ABB RAPID module: Mov.mod

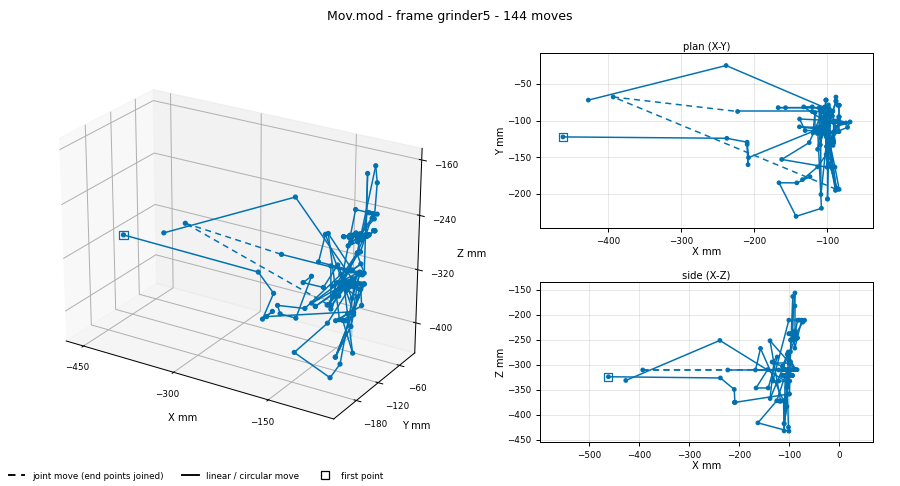
[picture p0: tool path of Mov.mod in frame grinder5, 144 of 396 moves have a stored position in this frame; points joined in program order, loops and branches not executed]
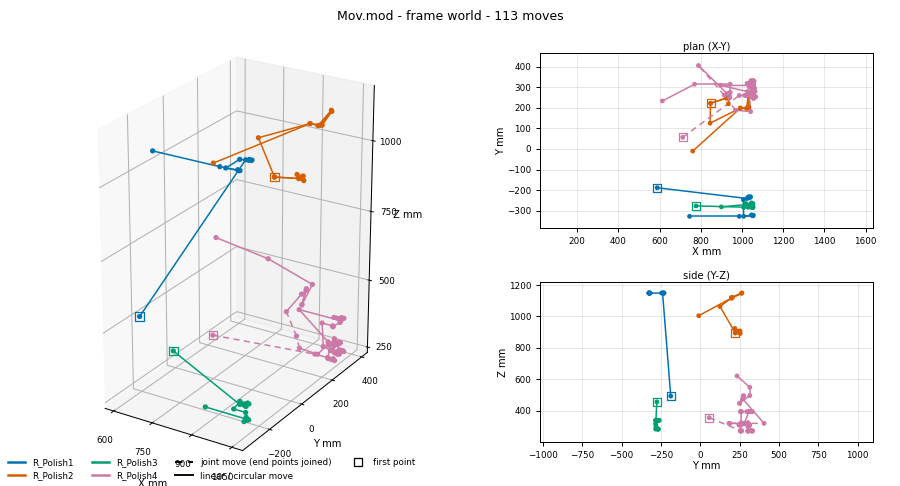
[picture p1: tool path of Mov.mod in frame world, 113 of 396 moves have a stored position in this frame; points joined in program order, loops and branches not executed]
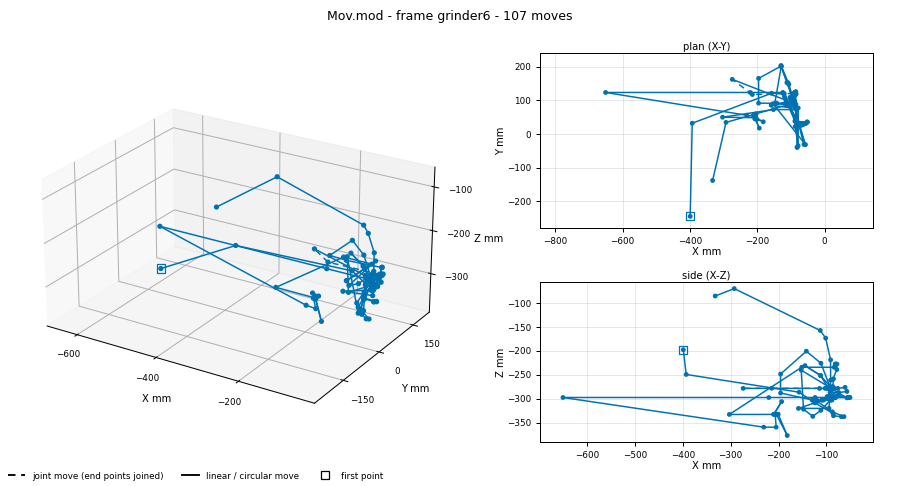
[picture p2: tool path of Mov.mod in frame grinder6, 107 of 396 moves have a stored position in this frame; points joined in program order, loops and branches not executed]
MODULE Mov

!******************************
! This program module for robot movements
! and storage of dynamic parameters
!******************************


! PALLET PARAMETERS
PERS num distance_p1_x:=60;
PERS num distance_p1_y:=160;
PERS num distance_p2_x:=60;
PERS num distance_p2_y:=160;

! DYNAMIC REGISTERS
PERS num loss_limit:=2;
PERS num collect:=1;
PERS num put:=1;
PERS num total:=0;
PERS num made:=0;
PERS num lost:=0;
PERS string start_data:="0000-00-00";

! TOOL DATA
PERS tooldata tool1:=[TRUE,[[0,0,320],[1,0,0,0]],[3,[0,0,130],[1,0,0,0],0,0,0]];
PERS tooldata tool2:=[TRUE,[[0,0,102],[1,0,0,0]],[3,[0,0,130],[1,0,0,0],0,0,0]];

TASK PERS tooldata a1:=[TRUE,[[0,0,344.1],[1,0,0,0]],[3,[0,0,130],[1,0,0,0],0,0,0]];
TASK PERS tooldata a2:=[TRUE,[[-72.3686,17.367,344.174],[1,0,0,0]],[3,[0,0,130],[1,0,0,0],0,0,0]];
TASK PERS tooldata a3:=[TRUE,[[-122,-5,344.174],[1,0,0,0]],[3,[0,0,130],[1,0,0,0],0,0,0]];
TASK PERS tooldata b1:=[TRUE,[[291.284,21.2677,171.248],[1,0,0,0]],[3,[70,0,130],[1,0,0,0],0,0,0]];

! WORK OBJECT DATA
PERS wobjdata pal1:=[FALSE,TRUE,"",[[760,-960,318],[4.81746E-05,-0.00506553,0.000941855,-0.999987]],[[540,0,0],[1,-9.27899E-07,1.32587E-06,-5.97185E-07]]];
PERS wobjdata pal2:=[FALSE,TRUE,"",[[149,-1059.8,461],[3.46326E-05,0.000526209,-0.000948043,0.999999]],[[0,0,0],[1,-3.72475E-06,5.79944E-06,-6.55528E-06]]];

TASK PERS wobjdata grinder1:=[FALSE,TRUE,"",[[1160.6,-280,1459],[1,0,0,0]],[[0,0,0],[1,0,0,0]]];
TASK PERS wobjdata grinder2:=[FALSE,TRUE,"",[[1160,280,1460],[1,0,0,0]],[[0,0,0],[1,0,0,0]]];
TASK PERS wobjdata grinder3:=[FALSE,TRUE,"",[[1156.5,-280,660],[1,0,0,0]],[[0,0,0],[1,0,0,0]]];
TASK PERS wobjdata grinder4:=[FALSE,TRUE,"",[[1158,280,656],[1,0,0,0]],[[6.65,0,-130],[1,0,0,0]]];
TASK PERS wobjdata grinder4_s:=[FALSE,TRUE,"",[[1157.8,510,518],[1,0,0,0]],[[0,0,0],[1,0,0,0]]];
TASK PERS wobjdata grinder5:=[FALSE,TRUE,"",[[280,1012,900],[0.70711,0,0,0.70711]],[[0,0,0],[1,0,0,0]]];
TASK PERS wobjdata grinder6:=[FALSE,TRUE,"",[[-282,1000,900],[0.70711,0,0,0.70711]],[[0,0,0],[1,0,0,0]]];

! POSITIONS
PERS robtarget home:=[[649.18,-0.03,789.42],[2.73078E-05,2.31734E-05,1,2.09338E-05],[-1,0,-1,0],[9E+09,9E+09,9E+09,9E+09,9E+09,9E+09]];
PERS robtarget corner:=[[286.64,-742.95,588.29],[0.00624253,-0.703358,-0.710805,0.00220458],[-1,-1,0,0],[9E+09,9E+09,9E+09,9E+09,9E+09,9E+09]];
PERS robtarget before:=[[683.43,-725.72,546.02],[0.0245473,-0.706641,-0.706937,-0.0172306],[-1,0,0,0],[9E+09,9E+09,9E+09,9E+09,9E+09,9E+09]];
PERS robtarget check:=[[764.25,-750.95,502.27],[0.0244543,-0.706556,-0.707026,-0.017169],[-1,0,0,0],[9E+09,9E+09,9E+09,9E+09,9E+09,9E+09]];
PERS robtarget after:=[[683.45,-725.70,546.02],[0.0245494,-0.706651,-0.706925,-0.0172644],[-1,0,0,0],[9E+09,9E+09,9E+09,9E+09,9E+09,9E+09]];
PERS robtarget non_drop:=[[286.65,-1103.34,974.46],[0.311182,0.630793,0.633652,-0.322103],[-1,-1,0,0],[9E+9,9E+9,9E+9,9E+9,9E+9,9E+9]];

PERS robtarget wheel5:=[[-112.72,-79.92,-299.81],[0.228521,0.250847,0.938723,-0.0604406],[0,-1,0,0],[9E+09,9E+09,9E+09,9E+09,9E+09,9E+09]];
PERS robtarget wheel6:=[[-100.57,98.49,-299.81],[0.221539,0.223786,0.947859,0.0490301],[1,-1,0,0],[9E+09,9E+09,9E+09,9E+09,9E+09,9E+09]];

! OFFSET PARAMETER
PERS num count5:=0;
PERS num count6:=0;
PERS num count5_limit:=1700;
PERS num count6_limit:=1700;

PERS num offs5_step:=0.01;
PERS num offs6_step:=0.01;


!******************************
PROC P_Parameters()
    distance_p1_x:=60;
    distance_p1_y:=160;
    distance_p2_x:=60;
    distance_p2_y:=160;
ENDPROC

!******************************
PROC R_Take1()
    Set DO10_60;
    !
    MoveL [[81.54,-63.78,264.56],[0.00371365,0.713716,-0.700414,0.00397575],[-1,-1,0,0],[9E+09,9E+09,9E+09,9E+09,9E+09,9E+09]],s500,z50,tool1\WObj:=pal1;
    MoveL [[79.44,-63.69,183.91],[0.011189,0.710235,-0.703782,0.0114969],[-1,0,0,0],[9E+09,9E+09,9E+09,9E+09,9E+09,9E+09]],s100,z10,tool1\WObj:=pal1;
    MoveL [[80.22,-63.55,118.78],[0.00697535,0.710341,-0.703813,0.00376915],[-1,0,0,0],[9E+09,9E+09,9E+09,9E+09,9E+09,9E+09]],s50,fine,tool1\WObj:=pal1;
    MoveL [[78.90,-63.58,118.50],[0.0118877,0.702177,-0.71189,-0.00426993],[-1,0,0,0],[9E+09,9E+09,9E+09,9E+09,9E+09,9E+09]],s25,fine,tool1\WObj:=pal1;
    MoveL [[78.90,-63.55,117.64],[0.00382538,0.726156,-0.687509,0.00387196],[-1,-1,0,0],[9E+09,9E+09,9E+09,9E+09,9E+09,9E+09]],s25,fine,tool1\WObj:=pal1;
    MoveL [[80.70,-63.58,116.47],[0.00384294,0.724898,-0.688834,0.00390763],[-1,-1,0,0],[9E+09,9E+09,9E+09,9E+09,9E+09,9E+09]],s25,fine,tool1\WObj:=pal1;
    !
    T_Grab;
    !
    MoveL [[81.00,-63.59,147.58],[0.0127632,0.716524,-0.697325,0.0129917],[-1,0,0,0],[9E+09,9E+09,9E+09,9E+09,9E+09,9E+09]],s50,fine,tool1\WObj:=pal1;
    MoveL [[81.31,-63.65,178.40],[0.0171099,0.716402,-0.69726,0.0174624],[-1,0,0,0],[9E+09,9E+09,9E+09,9E+09,9E+09,9E+09]],s150,z5,tool1\WObj:=pal1;
    MoveL [[81.48,-63.80,264.59],[0.00373939,0.713705,-0.700425,0.00394878],[-1,-1,0,0],[9E+09,9E+09,9E+09,9E+09,9E+09,9E+09]],s500,z50,tool1\WObj:=pal1;
ENDPROC

!******************************
PROC R_Take2()
    MoveL [[81.54,-63.78,264.56],[0.00371365,0.713716,-0.700414,0.00397575],[-1,-1,0,0],[9E+09,9E+09,9E+09,9E+09,9E+09,9E+09]],s500,z50,tool1\WObj:=pal1;
    MoveL [[79.44,-63.69,183.91],[0.011189,0.710235,-0.703782,0.0114969],[-1,0,0,0],[9E+09,9E+09,9E+09,9E+09,9E+09,9E+09]],s100,z10,tool1\WObj:=pal1;
    MoveL [[80.22,-63.55,118.78],[0.00697535,0.710341,-0.703813,0.00376915],[-1,0,0,0],[9E+09,9E+09,9E+09,9E+09,9E+09,9E+09]],s50,fine,tool1\WObj:=pal1;
    MoveL [[78.90,-63.58,118.50],[0.0118877,0.702177,-0.71189,-0.00426993],[-1,0,0,0],[9E+09,9E+09,9E+09,9E+09,9E+09,9E+09]],s25,fine,tool1\WObj:=pal1;
    MoveL [[78.90,-63.55,117.64],[0.00382538,0.726156,-0.687509,0.00387196],[-1,-1,0,0],[9E+09,9E+09,9E+09,9E+09,9E+09,9E+09]],s25,fine,tool1\WObj:=pal1;
    MoveL [[80.70,-63.58,116.47],[0.00384294,0.724898,-0.688834,0.00390763],[-1,-1,0,0],[9E+09,9E+09,9E+09,9E+09,9E+09,9E+09]],s25,fine,tool1\WObj:=pal1;
    !
    T_Grab;
    !
    MoveL [[81.00,-63.59,147.58],[0.0127632,0.716524,-0.697325,0.0129917],[-1,0,0,0],[9E+09,9E+09,9E+09,9E+09,9E+09,9E+09]],s50,fine,tool1\WObj:=pal1;
    MoveL [[81.31,-63.65,178.40],[0.0171099,0.716402,-0.69726,0.0174624],[-1,0,0,0],[9E+09,9E+09,9E+09,9E+09,9E+09,9E+09]],s150,z5,tool1\WObj:=pal1;
    MoveL [[81.48,-63.80,264.59],[0.00373939,0.713705,-0.700425,0.00394878],[-1,-1,0,0],[9E+09,9E+09,9E+09,9E+09,9E+09,9E+09]],s500,z50,tool1\WObj:=pal1;
ENDPROC

!******************************
PROC R_Drop1()
    MoveL [[81.49,-63.80,264.52],[0.00378181,0.713658,-0.700473,0.0039678],[-1,-1,0,0],[9E+09,9E+09,9E+09,9E+09,9E+09,9E+09]],s500,z50,tool1\WObj:=pal1;
    MoveL [[81.16,-63.64,177.38],[0.015051,0.720309,-0.693317,0.0154864],[-1,0,0,0],[9E+09,9E+09,9E+09,9E+09,9E+09,9E+09]],s500,z10,tool1\WObj:=pal1;
    MoveL [[80.98,-63.98,149.80],[0.0150862,0.715998,-0.697765,0.0155745],[-1,0,0,0],[9E+09,9E+09,9E+09,9E+09,9E+09,9E+09]],s100,z1,tool1\WObj:=pal1;
    MoveL [[79.99,-63.75,138.99],[0.0152028,0.720859,-0.692742,0.0154934],[-1,0,0,0],[9E+09,9E+09,9E+09,9E+09,9E+09,9E+09]],s50,fine,tool1\WObj:=pal1;
    !
    T_Release;
    !
    MoveL [[80.08,-63.90,158.90],[0.0175743,0.722459,-0.690952,0.0181282],[-1,0,0,0],[9E+09,9E+09,9E+09,9E+09,9E+09,9E+09]],s20,fine,tool1\WObj:=pal1;
    MoveL [[81.01,-63.73,207.27],[0.00381861,0.72049,-0.693443,0.00397601],[-1,-1,0,0],[9E+09,9E+09,9E+09,9E+09,9E+09,9E+09]],s50,z50,tool1\WObj:=pal1;
    MoveL [[81.54,-63.77,264.48],[0.00376586,0.713646,-0.700485,0.00398274],[-1,-1,0,0],[9E+09,9E+09,9E+09,9E+09,9E+09,9E+09]],s500,z50,tool1\WObj:=pal1;
    !
    Reset DO10_60;
ENDPROC

!******************************
PROC R_Drop2()
    MoveL [[81.49,-63.80,264.52],[0.00378181,0.713658,-0.700473,0.0039678],[-1,-1,0,0],[9E+09,9E+09,9E+09,9E+09,9E+09,9E+09]],s500,z50,tool1\WObj:=pal1;
    MoveL [[81.16,-63.64,177.38],[0.015051,0.720309,-0.693317,0.0154864],[-1,0,0,0],[9E+09,9E+09,9E+09,9E+09,9E+09,9E+09]],s500,z10,tool1\WObj:=pal1;
    MoveL [[80.98,-63.98,149.80],[0.0150862,0.715998,-0.697765,0.0155745],[-1,0,0,0],[9E+09,9E+09,9E+09,9E+09,9E+09,9E+09]],s100,z1,tool1\WObj:=pal1;
    MoveL [[79.99,-63.75,138.99],[0.0152028,0.720859,-0.692742,0.0154934],[-1,0,0,0],[9E+09,9E+09,9E+09,9E+09,9E+09,9E+09]],s50,fine,tool1\WObj:=pal1;
    !
    T_Release;
    !
    MoveL [[80.08,-63.90,158.90],[0.0175743,0.722459,-0.690952,0.0181282],[-1,0,0,0],[9E+09,9E+09,9E+09,9E+09,9E+09,9E+09]],s20,fine,tool1\WObj:=pal1;
    MoveL [[81.01,-63.73,207.27],[0.00381861,0.72049,-0.693443,0.00397601],[-1,-1,0,0],[9E+09,9E+09,9E+09,9E+09,9E+09,9E+09]],s50,z50,tool1\WObj:=pal1;
    MoveL [[81.54,-63.77,264.48],[0.00376586,0.713646,-0.700485,0.00398274],[-1,-1,0,0],[9E+09,9E+09,9E+09,9E+09,9E+09,9E+09]],s500,z50,tool1\WObj:=pal1;
    !
    Reset DO10_60;
ENDPROC

!******************************
PROC R_Polish1()
    MoveL [[-571.75,91.90,-965.06],[0.469276,0.555052,-0.658028,0.196717],[0,-1,-1,0],[9E+09,9E+09,9E+09,9E+09,9E+09,9E+09]],s800,z50,tool1\WObj:=grinder1;
    !
    T_RotateX;
    !
    MoveL [[-136.64,39.89,-310.14],[0.596711,0.562615,-0.456705,0.344705],[0,-1,-1,0],[9E+09,9E+09,9E+09,9E+09,9E+09,9E+09]],s500,z50,b1\WObj:=grinder1;
    !
    FOR i FROM 1 TO 2 DO
        MoveL [[-119.31,48.42,-310.14],[0.596621,0.562523,-0.456828,0.344847],[0,-1,-1,0],[9E+09,9E+09,9E+09,9E+09,9E+09,9E+09]],s100,z15,b1\WObj:=grinder1;
        MoveL [[-128.71,48.31,-310.17],[0.462741,0.446288,-0.567706,0.514206],[0,-1,-1,0],[9E+09,9E+09,9E+09,9E+09,9E+09,9E+09]],s100,z15,b1\WObj:=grinder1;
        MoveL [[-127.40,42.33,-310.13],[0.369211,0.463358,-0.680274,0.431521],[0,-1,-1,0],[9E+09,9E+09,9E+09,9E+09,9E+09,9E+09]],s100,z15,b1\WObj:=grinder1;
        MoveL [[-120.11,45.43,-310.13],[0.525624,0.633918,-0.444547,0.352484],[0,-1,-1,0],[9E+09,9E+09,9E+09,9E+09,9E+09,9E+09]],s100,z15,b1\WObj:=grinder1;
    ENDFOR
    !
    MoveL [[-153.60,33.89,-310.10],[0.525638,0.633914,-0.444522,0.352502],[0,-1,-1,0],[9E+09,9E+09,9E+09,9E+09,9E+09,9E+09]],s500,z50,b1\WObj:=grinder1;
    MoveL [[-152.18,-46.75,-310.15],[0.448349,0.726289,-0.37062,0.366234],[-1,-1,-2,0],[9E+09,9E+09,9E+09,9E+09,9E+09,9E+09]],s500,z50,b1\WObj:=grinder1;
    !
    !! Warning! Engine starting
    S_Grinder4 "Start";
    !!
    FOR i FROM 1 TO 2 DO
        MoveL [[-107.15,-44.37,-310.09],[0.418549,0.695255,-0.42594,0.400016],[-1,-1,-1,0],[9E+09,9E+09,9E+09,9E+09,9E+09,9E+09]],s100,z15,b1\WObj:=grinder1;
        MoveL [[-114.46,-39.82,-310.24],[0.245454,0.539907,-0.638209,0.490859],[0,-1,-1,0],[9E+09,9E+09,9E+09,9E+09,9E+09,9E+09]],s100,z15,b1\WObj:=grinder1;
        MoveL [[-110.87,-42.28,-310.27],[0.234933,0.626957,-0.599794,0.438154],[0,-1,-1,0],[9E+09,9E+09,9E+09,9E+09,9E+09,9E+09]],s100,z15,b1\WObj:=grinder1;
        MoveL [[-105.52,-41.38,-310.25],[0.343308,0.697221,-0.478669,0.408532],[0,-1,-1,0],[9E+09,9E+09,9E+09,9E+09,9E+09,9E+09]],s100,z15,b1\WObj:=grinder1;
    ENDFOR
    !
    MoveL [[-173.16,-46.87,-310.39],[0.356815,0.753084,-0.401612,0.37981],[-1,-1,-2,0],[9E+09,9E+09,9E+09,9E+09,9E+09,9E+09]],s500,z50,b1\WObj:=grinder1;
    MoveL [[-414.58,-46.87,-310.28],[0.409761,0.602765,-0.550529,0.407049],[0,-1,-1,0],[9E+09,9E+09,9E+09,9E+09,9E+09,9E+09]],s500,z200,b1\WObj:=grinder1;
    !!
    S_Grinder1 "Stop";
ENDPROC

!******************************
PROC R_Polish2()
    MoveL [[-312.18,-58.03,-564.65],[0.0659927,-0.213903,0.974446,0.0185996],[0,0,-1,0],[9E+09,9E+09,9E+09,9E+09,9E+09,9E+09]],s800,z50,tool1\WObj:=grinder2;
    !
    MoveL [[-234.88,-32.80,-561.97],[0.0656619,-0.204066,0.976564,0.0192098],[0,0,-1,0],[9E+09,9E+09,9E+09,9E+09,9E+09,9E+09]],s500,z50,tool1\WObj:=grinder2;
    MoveL [[-220.20,-26.41,-568.20],[0.0654639,-0.195529,0.978311,0.0197588],[0,0,-1,0],[9E+09,9E+09,9E+09,9E+09,9E+09,9E+09]],s100,fine,tool1\WObj:=grinder2;
    MoveL [[-225.85,-60.76,-535.94],[0.0654396,-0.19553,0.978313,0.0197444],[0,0,-1,0],[9E+09,9E+09,9E+09,9E+09,9E+09,9E+09]],s100,fine,tool1\WObj:=grinder2;
    MoveL [[-222.19,-27.42,-552.18],[0.0654156,-0.195537,0.978313,0.0197604],[0,0,-1,0],[9E+09,9E+09,9E+09,9E+09,9E+09,9E+09]],s100,fine,tool1\WObj:=grinder2;
    MoveL [[-234.88,-32.80,-561.97],[0.0656619,-0.204066,0.976564,0.0192098],[0,0,-1,0],[9E+09,9E+09,9E+09,9E+09,9E+09,9E+09]],s500,z50,tool1\WObj:=grinder2;
    !
    MoveL [[-312.18,-58.03,-564.65],[0.0659927,-0.213903,0.974446,0.0185996],[0,0,-1,0],[9E+09,9E+09,9E+09,9E+09,9E+09,9E+09]],s500,z50,tool1\WObj:=grinder2;
    !
    MoveL [[-314.79,-154.83,-396.62],[0.493585,-0.336846,0.701772,-0.387846],[0,-1,0,0],[9E+9,9E+9,9E+9,9E+9,9E+9,9E+9]],s500,z50,tool1\WObj:=grinder2;
    MoveL [[-167.92,-81.52,-342.31],[0.588966,-0.355549,0.620647,-0.376166],[0,-2,0,0],[9E+9,9E+9,9E+9,9E+9,9E+9,9E+9]],s500,z50,tool1\WObj:=grinder2;
    !
    !! Warning! Engine starting
    S_Grinder3 "Start";
    !!
    MoveL [[-138.04,-82.74,-343.00],[0.607835,-0.322275,0.598705,-0.410156],[0,-2,0,0],[9E+09,9E+09,9E+09,9E+09,9E+09,9E+09]],s100,fine,tool1\WObj:=grinder2;
    MoveL [[-128.40,-15.83,-310.47],[0.598332,-0.339516,0.610415,-0.392583],[0,-2,0,0],[9E+9,9E+9,9E+9,9E+9,9E+9,9E+9]],s100,fine,tool1\WObj:=grinder2;
    MoveL [[-127.12,-78.24,-340.07],[0.603187,-0.330919,0.604506,-0.401535],[0,-2,0,0],[9E+9,9E+9,9E+9,9E+9,9E+9,9E+9]],s100,fine,tool1\WObj:=grinder2;
    MoveL [[-126.22,-77.24,-340.26],[0.589644,-0.354395,0.619971,-0.377306],[0,-2,0,0],[9E+9,9E+9,9E+9,9E+9,9E+9,9E+9]],s50,fine,tool1\WObj:=grinder2;
    MoveL [[-125.00,-18.54,-312.77],[0.593442,-0.347907,0.615964,-0.383896],[0,-2,0,0],[9E+9,9E+9,9E+9,9E+9,9E+9,9E+9]],s100,fine,tool1\WObj:=grinder2;
    MoveL [[-130.31,-81.29,-340.25],[0.592287,-0.349923,0.617288,-0.381713],[0,-2,0,0],[9E+9,9E+9,9E+9,9E+9,9E+9,9E+9]],s100,fine,tool1\WObj:=grinder2;
    !
    MoveL [[-167.92,-81.52,-342.31],[0.588966,-0.355549,0.620647,-0.376166],[0,-2,0,0],[9E+9,9E+9,9E+9,9E+9,9E+9,9E+9]],s500,z50,tool1\WObj:=grinder2;
    MoveL [[-398.88,-290.20,-455.37],[0.408162,-0.140842,0.79461,-0.426806],[0,-1,0,0],[9E+09,9E+09,9E+09,9E+09,9E+09,9E+09]],s500,z50,tool1\WObj:=grinder2;
    !!
    S_Grinder2 "Stop";
ENDPROC

!******************************
PROC R_Polish3()
    MoveJ [[-379.07,3.77,-202.95],[0.683485,0.708062,-0.101976,0.145252],[0,-1,-2,0],[9E+09,9E+09,9E+09,9E+09,9E+09,9E+09]],s800,z50,tool1\WObj:=grinder3;
    MoveL [[-126.34,-2.73,-320.36],[0.68352,0.707981,-0.101962,0.145489],[0,-1,-2,0],[9E+09,9E+09,9E+09,9E+09,9E+09,9E+09]],s800,z50,tool1\WObj:=grinder3;
    !
    MoveL [[-103.08,-2.45,-320.45],[0.701277,0.704012,-0.0566479,0.0967937],[0,-1,-2,0],[9E+09,9E+09,9E+09,9E+09,9E+09,9E+09]],s100,fine,tool1\WObj:=grinder3;
    MoveL [[-104.83,-3.28,-320.38],[0.624078,0.640547,-0.297462,0.334278],[0,-1,-1,0],[9E+09,9E+09,9E+09,9E+09,9E+09,9E+09]],s100,z5,tool1\WObj:=grinder3;
    MoveL [[-106.41,-1.18,-320.42],[0.535858,0.497066,-0.395151,0.556451],[0,-2,-1,0],[9E+09,9E+09,9E+09,9E+09,9E+09,9E+09]],s100,z5,tool1\WObj:=grinder3;
    MoveL [[-110.93,2.25,-320.50],[0.00914576,0.0131634,-0.680054,0.732987],[0,-1,0,0],[9E+09,9E+09,9E+09,9E+09,9E+09,9E+09]],s100,z5,tool1\WObj:=grinder3;
    MoveL [[-118.21,4.22,-320.58],[0.0670865,-0.095308,0.682521,-0.721513],[0,-2,0,0],[9E+09,9E+09,9E+09,9E+09,9E+09,9E+09]],s50,z5,tool1\WObj:=grinder3;
    MoveL [[-114.81,7.39,-320.41],[0.257779,0.206079,-0.602722,0.726504],[0,-1,0,0],[9E+09,9E+09,9E+09,9E+09,9E+09,9E+09]],s100,z5,tool1\WObj:=grinder3;
    MoveL [[-110.51,18.54,-320.42],[0.435856,0.395761,-0.399732,0.702579],[0,-2,-1,0],[9E+09,9E+09,9E+09,9E+09,9E+09,9E+09]],s100,z5,tool1\WObj:=grinder3;
    MoveL [[-103.74,15.02,-320.44],[0.805324,0.562494,-0.00198576,0.187219],[0,-2,-2,0],[9E+09,9E+09,9E+09,9E+09,9E+09,9E+09]],s100,fine,tool1\WObj:=grinder3;
    !
    MoveL [[-137.02,14.99,-320.43],[0.808451,0.562444,0.00783305,0.173212],[0,-2,-2,0],[9E+09,9E+09,9E+09,9E+09,9E+09,9E+09]],s200,z50,tool1\WObj:=grinder3;
    !
    !! Warning! Engine starting
    S_Grinder1 "Start";
    !!
    MoveL [[-148.15,-3.78,-342.00],[0.66253,0.672145,0.260987,-0.202881],[0,-1,-2,0],[9E+09,9E+09,9E+09,9E+09,9E+09,9E+09]],s500,z50,tool1\WObj:=grinder3;
    MoveL [[-103.97,-3.77,-342.00],[0.662534,0.672142,0.260992,-0.202873],[0,-1,-2,0],[9E+09,9E+09,9E+09,9E+09,9E+09,9E+09]],s100,fine,tool1\WObj:=grinder3;
    MoveL [[-103.08,-2.17,-359.59],[0.567234,0.588951,0.463739,-0.34107],[0,-1,-3,0],[9E+09,9E+09,9E+09,9E+09,9E+09,9E+09]],s100,z5,tool1\WObj:=grinder3;
    MoveL [[-110.08,-3.78,-376.14],[0.35843,0.307487,0.75861,-0.448877],[0,-2,-3,0],[9E+09,9E+09,9E+09,9E+09,9E+09,9E+09]],s100,fine,tool1\WObj:=grinder3;
    MoveL [[-110.12,10.83,-376.16],[0.358414,0.307541,0.758609,-0.448855],[0,-1,-3,0],[9E+09,9E+09,9E+09,9E+09,9E+09,9E+09]],s50,fine,tool1\WObj:=grinder3;
    MoveL [[-107.10,8.56,-376.11],[0.556404,0.605548,0.467899,-0.323722],[0,-1,-3,0],[9E+09,9E+09,9E+09,9E+09,9E+09,9E+09]],s200,fine,tool1\WObj:=grinder3;
    MoveL [[-103.49,13.88,-376.18],[0.669728,0.646124,0.336954,-0.143004],[0,-2,-2,0],[9E+09,9E+09,9E+09,9E+09,9E+09,9E+09]],s100,z5,tool1\WObj:=grinder3;
    !
    MoveL [[-256.29,-1.00,-366.66],[0.677428,0.697554,0.180679,-0.14787],[0,-1,-2,0],[9E+09,9E+09,9E+09,9E+09,9E+09,9E+09]],s500,z50,tool1\WObj:=grinder3;
    !!
    S_Grinder3 "Stop";
ENDPROC

!******************************
PROC R_Polish4()
    MoveJ [[-452.02,-223.42,-169.43],[0.436016,-0.54839,0.445538,0.557364],[-1,0,-2,0],[9E+09,9E+09,9E+09,9E+09,9E+09,9E+09]],s500,z200,b1\WObj:=grinder4;
    !
    MoveJ [[-177.43,-20.14,-253.32],[0.612772,-0.788995,0.0279635,0.0348631],[0,0,-3,0],[9E+09,9E+09,9E+09,9E+09,9E+09,9E+09]],s500,z50,b1\WObj:=grinder4;
    MoveL [[-128.24,-20.11,-253.35],[0.612409,-0.789344,0.0351394,0.0256267],[0,0,-3,0],[9E+09,9E+09,9E+09,9E+09,9E+09,9E+09]],s300,z50,b1\WObj:=grinder4;
    !
    MoveL [[-97.45,-26.65,-253.35],[0.611663,-0.788717,-0.0479453,-0.0386689],[0,0,-3,0],[9E+09,9E+09,9E+09,9E+09,9E+09,9E+09]],s100,z5,b1\WObj:=grinder4;
    MoveL [[-109.41,-25.52,-253.38],[0.567279,-0.663532,0.336259,0.35334],[0,0,-2,0],[9E+09,9E+09,9E+09,9E+09,9E+09,9E+09]],s100,z5,b1\WObj:=grinder4;
    MoveL [[-108.27,-17.16,-253.35],[0.492481,-0.487886,0.413521,0.59028],[-1,0,-2,0],[9E+09,9E+09,9E+09,9E+09,9E+09,9E+09]],s100,z5,b1\WObj:=grinder4;
    MoveL [[-121.23,-24.09,-253.34],[0.284698,-0.284928,0.566027,0.719289],[-1,1,-2,0],[9E+09,9E+09,9E+09,9E+09,9E+09,9E+09]],s100,z5,b1\WObj:=grinder4;
    MoveL [[-124.32,-24.11,-253.36],[0.108741,-0.169556,0.70879,0.67605],[0,0,-1,0],[9E+09,9E+09,9E+09,9E+09,9E+09,9E+09]],s100,z5,b1\WObj:=grinder4;
    MoveL [[-119.24,-21.33,-200.73],[0.00771246,0.0104736,-0.724419,-0.689237],[0,0,-1,0],[9E+09,9E+09,9E+09,9E+09,9E+09,9E+09]],s100,z5,b1\WObj:=grinder4;
    !
    MoveL [[-127.47,22.43,-200.63],[0.00773932,0.0103727,-0.724355,-0.689305],[0,0,-1,0],[9E+09,9E+09,9E+09,9E+09,9E+09,9E+09]],s100,z5,b1\WObj:=grinder4;
    MoveL [[-129.72,22.83,-226.68],[0.137614,-0.100798,0.660326,0.731349],[0,1,-1,0],[9E+09,9E+09,9E+09,9E+09,9E+09,9E+09]],s100,z5,b1\WObj:=grinder4;
    MoveL [[-126.92,23.02,-253.07],[0.279621,-0.188828,0.572046,0.747609],[0,1,-1,0],[9E+09,9E+09,9E+09,9E+09,9E+09,9E+09]],s100,z5,b1\WObj:=grinder4;
    MoveL [[-123.69,23.08,-253.17],[0.403833,-0.314025,0.506286,0.69425],[-1,1,-2,0],[9E+09,9E+09,9E+09,9E+09,9E+09,9E+09]],s100,z5,b1\WObj:=grinder4;
    MoveL [[-114.51,23.26,-255.31],[0.570642,-0.474681,0.398583,0.538681],[-1,1,-2,0],[9E+09,9E+09,9E+09,9E+09,9E+09,9E+09]],s100,z5,b1\WObj:=grinder4;
    MoveL [[-113.12,22.82,-253.71],[0.675504,-0.647991,0.235961,0.261005],[0,1,-3,0],[9E+09,9E+09,9E+09,9E+09,9E+09,9E+09]],s100,z5,b1\WObj:=grinder4;
    MoveL [[-107.64,22.86,-253.66],[0.733343,-0.678622,-0.0244374,-0.0329145],[0,1,-3,0],[9E+09,9E+09,9E+09,9E+09,9E+09,9E+09]],s100,z5,b1\WObj:=grinder4;
    !
    MoveL [[-105.02,48.26,-253.70],[0.732639,-0.67849,-0.041679,-0.0339785],[0,1,-3,0],[9E+09,9E+09,9E+09,9E+09,9E+09,9E+09]],s100,z5,b1\WObj:=grinder4;
    MoveL [[-110.61,52.72,-253.63],[0.706933,-0.583588,0.288358,0.276624],[0,1,-3,0],[9E+09,9E+09,9E+09,9E+09,9E+09,9E+09]],s100,z5,b1\WObj:=grinder4;
    MoveL [[-115.77,45.83,-253.63],[0.7317,-0.41417,0.297486,0.452306],[-1,1,-2,0],[9E+09,9E+09,9E+09,9E+09,9E+09,9E+09]],s100,z5,b1\WObj:=grinder4;
    MoveL [[-121.21,51.75,-253.65],[0.588482,-0.322299,0.395175,0.627414],[-1,1,-2,0],[9E+09,9E+09,9E+09,9E+09,9E+09,9E+09]],s100,z5,b1\WObj:=grinder4;
    MoveL [[-122.73,43.06,-253.64],[0.52963,-0.285341,0.422601,0.67785],[-1,1,-2,0],[9E+09,9E+09,9E+09,9E+09,9E+09,9E+09]],s100,z5,b1\WObj:=grinder4;
    MoveL [[-121.67,33.01,-215.73],[0.404729,-0.210891,0.49619,0.73859],[-1,1,-2,0],[9E+09,9E+09,9E+09,9E+09,9E+09,9E+09]],s100,z5,b1\WObj:=grinder4;
    MoveL [[-127.01,21.46,-215.62],[0.23649,-0.142846,0.582942,0.764098],[0,1,-1,0],[9E+09,9E+09,9E+09,9E+09,9E+09,9E+09]],s100,z5,b1\WObj:=grinder4;
    MoveL [[-111.94,30.40,-215.60],[0.00647471,-0.0298945,0.683911,0.728924],[0,1,-1,0],[9E+09,9E+09,9E+09,9E+09,9E+09,9E+09]],s100,z5,b1\WObj:=grinder4;
    MoveL [[-109.38,-28.50,-215.64],[0.00645724,-0.029982,0.683965,0.72887],[0,1,-1,0],[9E+09,9E+09,9E+09,9E+09,9E+09,9E+09]],s50,z5,b1\WObj:=grinder4;
    MoveL [[-110.37,32.89,-215.55],[0.00216545,0.0390885,-0.683974,-0.728455],[0,1,-1,0],[9E+09,9E+09,9E+09,9E+09,9E+09,9E+09]],s50,z5,b1\WObj:=grinder4;
    MoveL [[-108.23,-34.29,-215.67],[0.0101001,-0.0259263,0.684008,0.728943],[-1,1,-1,0],[9E+09,9E+09,9E+09,9E+09,9E+09,9E+09]],s50,z5,b1\WObj:=grinder4;
    MoveL [[-110.37,32.89,-215.55],[0.00216545,0.0390885,-0.683974,-0.728455],[0,1,-1,0],[9E+09,9E+09,9E+09,9E+09,9E+09,9E+09]],s50,z5,b1\WObj:=grinder4;
    MoveL [[-108.23,-34.29,-215.67],[0.0101001,-0.0259263,0.684008,0.728943],[-1,1,-1,0],[9E+09,9E+09,9E+09,9E+09,9E+09,9E+09]],s50,z5,b1\WObj:=grinder4;
    MoveL [[-144.60,-21.59,-215.64],[0.00374565,-0.0277671,0.691645,0.721694],[0,1,-1,0],[9E+09,9E+09,9E+09,9E+09,9E+09,9E+09]],s200,z5,b1\WObj:=grinder4;
    !
    MoveL [[-151.64,-19.83,-131.15],[0.198108,-0.282286,-0.630265,-0.695581],[-1,1,-1,0],[9E+09,9E+09,9E+09,9E+09,9E+09,9E+09]],s300,z50,b1\WObj:=grinder4;
    !
    MoveL [[-111.43,-19.84,-131.13],[0.198113,-0.282307,-0.630236,-0.695598],[-1,1,-1,0],[9E+09,9E+09,9E+09,9E+09,9E+09,9E+09]],s100,z5,b1\WObj:=grinder4;
    MoveL [[-106.49,-24.53,-131.13],[0.349117,-0.583677,-0.429742,-0.593936],[0,1,0,0],[9E+09,9E+09,9E+09,9E+09,9E+09,9E+09]],s100,z5,b1\WObj:=grinder4;
    MoveL [[-107.96,-24.54,-131.12],[0.568957,-0.654369,-0.215527,-0.449041],[0,1,0,0],[9E+09,9E+09,9E+09,9E+09,9E+09,9E+09]],s100,z5,b1\WObj:=grinder4;
    MoveL [[-103.29,14.99,-131.09],[0.528927,-0.656326,-0.406016,-0.35302],[-1,0,0,0],[9E+09,9E+09,9E+09,9E+09,9E+09,9E+09]],s100,z5,b1\WObj:=grinder4;
    MoveL [[-107.93,28.60,-131.08],[0.226248,-0.230524,-0.754036,-0.571926],[0,0,-1,0],[9E+09,9E+09,9E+09,9E+09,9E+09,9E+09]],s100,z5,b1\WObj:=grinder4;
    MoveL [[-107.96,28.57,-131.13],[0.31549,-0.366512,-0.742769,-0.463066],[-1,0,0,0],[9E+09,9E+09,9E+09,9E+09,9E+09,9E+09]],s100,z5,b1\WObj:=grinder4;
    MoveL [[-119.79,40.20,-131.11],[0.289164,-0.54426,-0.769469,-0.167578],[-1,0,0,0],[9E+09,9E+09,9E+09,9E+09,9E+09,9E+09]],s100,z5,b1\WObj:=grinder4;
    MoveL [[-139.55,38.36,-131.14],[0.402812,-0.620744,-0.669778,0.0617797],[-1,0,0,0],[9E+09,9E+09,9E+09,9E+09,9E+09,9E+09]],s100,z5,b1\WObj:=grinder4;
    MoveL [[-127.79,38.36,-131.15],[0.401293,-0.697887,-0.592649,-0.026161],[-1,0,0,0],[9E+09,9E+09,9E+09,9E+09,9E+09,9E+09]],s100,z5,b1\WObj:=grinder4;
    MoveL [[-117.13,49.87,-131.11],[0.517937,-0.630929,-0.545499,-0.190003],[-1,0,0,0],[9E+09,9E+09,9E+09,9E+09,9E+09,9E+09]],s100,z5,b1\WObj:=grinder4;
    MoveL [[-107.98,49.89,-131.14],[0.410037,-0.590452,-0.625958,-0.302345],[-1,0,0,0],[9E+09,9E+09,9E+09,9E+09,9E+09,9E+09]],s100,z5,b1\WObj:=grinder4;
    MoveL [[-107.93,28.55,-131.12],[0.650239,-0.560619,-0.391377,-0.33124],[0,0,0,0],[9E+09,9E+09,9E+09,9E+09,9E+09,9E+09]],s100,z5,b1\WObj:=grinder4;
    !
    MoveL [[-268.49,28.57,-131.17],[0.602904,-0.59384,-0.461107,-0.266911],[-1,0,0,0],[9E+09,9E+09,9E+09,9E+09,9E+09,9E+09]],s500,z50,b1\WObj:=grinder4;
    !
    T_RotateZ;
    !
    MoveL [[-137.91,-1.01,-205.45],[0.715172,-0.689966,0.102725,0.043855],[-1,0,1,0],[9E+09,9E+09,9E+09,9E+09,9E+09,9E+09]],s800,z50,tool1\WObj:=grinder4;
    !
    MoveL [[-113.58,-1.02,-205.43],[0.715188,-0.689953,0.102716,0.0438206],[-1,0,1,0],[9E+09,9E+09,9E+09,9E+09,9E+09,9E+09]],s100,z5,tool1\WObj:=grinder4;
    MoveL [[-110.93,3.33,-205.43],[0.552628,-0.649139,0.449031,0.267568],[-1,0,2,0],[9E+09,9E+09,9E+09,9E+09,9E+09,9E+09]],s100,z5,tool1\WObj:=grinder4;
    MoveL [[-110.94,-1.09,-205.44],[0.394374,-0.568539,0.645957,0.322449],[-1,0,2,0],[9E+09,9E+09,9E+09,9E+09,9E+09,9E+09]],s100,z5,tool1\WObj:=grinder4;
    MoveL [[-110.97,-9.11,-205.48],[0.455866,-0.674064,0.579125,0.0493716],[-1,1,2,0],[9E+09,9E+09,9E+09,9E+09,9E+09,9E+09]],s100,z5,tool1\WObj:=grinder4;
    MoveL [[-100.80,-0.86,-205.49],[0.757534,-0.635358,0.0909885,0.119095],[-1,0,1,0],[9E+09,9E+09,9E+09,9E+09,9E+09,9E+09]],s100,z5,tool1\WObj:=grinder4;
    MoveL [[-128.30,-16.93,-205.61],[0.523363,-0.461535,0.561438,-0.44482],[0,2,1,0],[9E+09,9E+09,9E+09,9E+09,9E+09,9E+09]],s100,z5,tool1\WObj:=grinder4;
    MoveL [[-122.41,-98.59,-205.62],[0.52604,-0.463827,0.558787,-0.44261],[0,2,1,0],[9E+09,9E+09,9E+09,9E+09,9E+09,9E+09]],s50,z5,tool1\WObj:=grinder4;
    MoveL [[-195.59,-91.61,-205.59],[0.526101,-0.463704,0.558865,-0.442567],[0,2,1,0],[9E+09,9E+09,9E+09,9E+09,9E+09,9E+09]],s200,z5,tool1\WObj:=grinder4;
    !
    !! Warning! Engine starting
    S_Grinder5 "Start";
    !!
    MoveJ [[-249.60,-19.39,-205.62],[0.587569,-0.483279,0.508139,-0.40373],[0,2,1,0],[9E+09,9E+09,9E+09,9E+09,9E+09,9E+09]],s500,z50,tool1\WObj:=grinder4;
    !
    MoveJ [[-375.61,125.08,-205.66],[0.19782,-0.197359,0.652527,0.704362],[0,0,-2,0],[9E+09,9E+09,9E+09,9E+09,9E+09,9E+09]],s500,z50,tool1\WObj:=grinder4;
    !
    MoveL [[-236.63,-11.29,-49.62],[0.126276,-0.161831,0.708541,0.675155],[-1,0,-1,0],[9E+09,9E+09,9E+09,9E+09,9E+09,9E+09]],s500,z50,tool1\WObj:=grinder4;
    MoveL [[-222.78,-5.97,-34.88],[0.126473,-0.161935,0.708481,0.675156],[-1,0,-1,0],[9E+09,9E+09,9E+09,9E+09,9E+09,9E+09]],s100,z5,tool1\WObj:=grinder4;
    MoveL [[-224.13,-30.56,-78.81],[0.121095,-0.156619,0.709792,0.676019],[-1,0,-1,0],[9E+09,9E+09,9E+09,9E+09,9E+09,9E+09]],s100,z5,tool1\WObj:=grinder4;
    MoveL [[-221.98,-5.48,-28.66],[0.126337,-0.16203,0.708531,0.675107],[-1,0,-1,0],[9E+09,9E+09,9E+09,9E+09,9E+09,9E+09]],s100,z5,tool1\WObj:=grinder4;
    MoveL [[-223.51,-29.96,-77.26],[0.126195,-0.162023,0.708568,0.675096],[-1,0,-1,0],[9E+09,9E+09,9E+09,9E+09,9E+09,9E+09]],s100,z5,tool1\WObj:=grinder4;
    MoveL [[-222.00,34.28,-28.70],[0.126331,-0.162053,0.708545,0.675088],[-1,0,-1,0],[9E+09,9E+09,9E+09,9E+09,9E+09,9E+09]],s100,z5,tool1\WObj:=grinder4;
    !
    MoveL [[-394.77,34.28,23.97],[0.126342,-0.162103,0.708562,0.675056],[-1,0,-1,0],[9E+09,9E+09,9E+09,9E+09,9E+09,9E+09]],s500,z200,tool1\WObj:=grinder4;
    MoveL [[-550.86,-46.80,95.71],[0.0296238,0.21754,-0.975448,-0.0173241],[0,0,-1,0],[9E+09,9E+09,9E+09,9E+09,9E+09,9E+09]],s500,z50,tool1\WObj:=grinder4;
    !!
    S_Grinder4 "Stop";
ENDPROC

!******************************
PROC R_Polish5()
    P_OffsetCalculation 5;
    !
    S_WaxRed;
    !
    MoveL [[-461.20,-122.31,-324.13],[0.0659614,-0.206582,0.967604,-0.129286],[0,-1,-1,0],[9E+09,9E+09,9E+09,9E+09,9E+09,9E+09]],s500,z50,tool1\WObj:=grinder5;
    !
    MoveL [[-237.27,-124.18,-326.58],[0.0945029,-0.209766,0.963873,-0.134223],[0,-1,-1,0],[9E+09,9E+09,9E+09,9E+09,9E+09,9E+09]],s500,z50,tool1\WObj:=grinder5;
    !
    MoveL [[-209.53,-129.48,-349.44],[0.0944534,-0.209754,0.963881,-0.134219],[0,-1,-1,0],[9E+09,9E+09,9E+09,9E+09,9E+09,9E+09]],s100,z10,a1\WObj:=grinder5;
    MoveL [[-208.29,-160.16,-375.36],[0.0944539,-0.209734,0.963891,-0.134183],[0,-1,-1,0],[9E+09,9E+09,9E+09,9E+09,9E+09,9E+09]],s100,z10,a1\WObj:=grinder5;
    MoveL [[-209.44,-132.51,-375.38],[0.0944288,-0.20965,0.963915,-0.134157],[0,-1,-1,0],[9E+09,9E+09,9E+09,9E+09,9E+09,9E+09]],s100,z10,a1\WObj:=grinder5;
    MoveL [[-207.64,-150.49,-375.36],[0.0930947,-0.210375,0.964714,-0.128075],[0,-1,-1,0],[9E+09,9E+09,9E+09,9E+09,9E+09,9E+09]],s100,z10,a1\WObj:=grinder5;
    MoveL [[-100.25,-106.90,-358.67],[0.0200222,0.163036,-0.914206,0.370467],[0,-1,-1,0],[9E+09,9E+09,9E+09,9E+09,9E+09,9E+09]],s100,z10,a3\WObj:=grinder5;
    MoveL [[-98.97,-82.68,-358.67],[0.0197269,-0.0643179,0.926399,-0.370485],[0,-1,0,0],[9E+09,9E+09,9E+09,9E+09,9E+09,9E+09]],s100,z10,a3\WObj:=grinder5;
    MoveL [[-98.54,-87.11,-332.68],[0.0944388,-0.209734,0.963888,-0.134215],[0,-1,-1,0],[9E+09,9E+09,9E+09,9E+09,9E+09,9E+09]],s100,z10,a3\WObj:=grinder5;
    !
    MoveL [[-120.56,-81.31,-332.76],[0.0944925,-0.209714,0.963901,-0.134109],[0,-1,-1,0],[9E+09,9E+09,9E+09,9E+09,9E+09,9E+09]],s100,z50,a3\WObj:=grinder5;
    MoveL [[-132.22,-81.36,-332.65],[0.436128,0.587369,-0.365644,0.575408],[1,-2,-1,0],[9E+09,9E+09,9E+09,9E+09,9E+09,9E+09]],s200,z50,a3\WObj:=grinder5;
    !
    S_WaxRed;
    !
    MoveL [[-100.36,-103.25,-210.92],[0.484466,0.616939,-0.313259,0.535301],[1,-2,-1,0],[9E+09,9E+09,9E+09,9E+09,9E+09,9E+09]],s100,z50,a1\WObj:=grinder5;
    MoveL [[-79.47,-103.26,-210.94],[0.496095,0.623672,-0.299673,0.524518],[1,-2,-1,0],[9E+09,9E+09,9E+09,9E+09,9E+09,9E+09]],s50,z10,a1\WObj:=grinder5;
    MoveL [[-82.81,-103.25,-210.91],[0.557342,0.568403,-0.349183,0.494328],[1,-2,-1,0],[9E+09,9E+09,9E+09,9E+09,9E+09,9E+09]],s50,z10,a1\WObj:=grinder5;
    MoveL [[-90.66,-103.26,-250.78],[0.471724,0.609393,-0.327725,0.546546],[1,-2,-1,0],[9E+09,9E+09,9E+09,9E+09,9E+09,9E+09]],s50,z10,a1\WObj:=grinder5;
    MoveL [[-92.52,-87.29,-250.70],[0.13054,0.718651,-0.0666121,0.679752],[0,-3,0,0],[9E+09,9E+09,9E+09,9E+09,9E+09,9E+09]],s100,z10,a1\WObj:=grinder5;
    MoveL [[-92.51,-87.26,-163.61],[0.130574,0.718677,-0.0665137,0.679727],[0,-3,0,0],[9E+09,9E+09,9E+09,9E+09,9E+09,9E+09]],s100,z10,a1\WObj:=grinder5;
    MoveL [[-98.44,-78.76,-312.13],[0.142004,0.715351,-0.0765097,0.679893],[0,-3,-1,0],[9E+09,9E+09,9E+09,9E+09,9E+09,9E+09]],s100,z10,a1\WObj:=grinder5;
    MoveL [[-97.08,-102.61,-273.97],[0.0460851,0.72894,0.0128513,0.682904],[0,-3,0,0],[9E+09,9E+09,9E+09,9E+09,9E+09,9E+09]],s100,z10,a1\WObj:=grinder5;
    MoveL [[-88.15,-73.44,-156.51],[0.00716239,0.744496,0.0328827,0.666779],[0,-3,0,0],[9E+09,9E+09,9E+09,9E+09,9E+09,9E+09]],s100,z10,a1\WObj:=grinder5;
    MoveL [[-88.16,-67.97,-182.55],[0.00465908,0.746355,0.0330513,0.664711],[0,-3,0,0],[9E+09,9E+09,9E+09,9E+09,9E+09,9E+09]],s50,z10,a1\WObj:=grinder5;
    MoveL [[-88.16,-73.48,-232.49],[0.202689,0.718347,-0.144458,0.649636],[0,-2,-1,0],[9E+09,9E+09,9E+09,9E+09,9E+09,9E+09]],s100,z10,a1\WObj:=grinder5;
    !
    S_WaxRed;
    !
    MoveL [[-97.02,-102.67,-250.66],[0.487825,0.54545,-0.409899,0.544513],[1,-2,-1,0],[9E+09,9E+09,9E+09,9E+09,9E+09,9E+09]],s100,z10,a1\WObj:=grinder5;
    MoveL [[-94.15,-132.68,-250.65],[0.487844,0.545446,-0.409875,0.544517],[1,-2,-1,0],[9E+09,9E+09,9E+09,9E+09,9E+09,9E+09]],s50,z10,a1\WObj:=grinder5;
    MoveL [[-90.17,-114.40,-250.65],[0.727609,0.678993,0.0667965,0.0713555],[1,-2,-2,0],[9E+09,9E+09,9E+09,9E+09,9E+09,9E+09]],s100,z10,a1\WObj:=grinder5;
    MoveL [[-88.44,-109.02,-267.02],[0.726325,0.649866,0.0991701,0.200728],[0,-2,-2,0],[9E+09,9E+09,9E+09,9E+09,9E+09,9E+09]],s100,z10,a1\WObj:=grinder5;
    MoveL [[-74.60,-103.25,-210.92],[0.496105,0.623671,-0.299634,0.524532],[1,-2,-1,0],[9E+09,9E+09,9E+09,9E+09,9E+09,9E+09]],s100,z10,a1\WObj:=grinder5;
    MoveL [[-68.92,-101.81,-210.98],[0.536209,0.769211,0.0220081,0.346857],[0,-2,-2,0],[9E+09,9E+09,9E+09,9E+09,9E+09,9E+09]],s100,z10,a1\WObj:=grinder5;
    MoveL [[-72.34,-109.28,-214.82],[0.661492,0.647031,-0.129382,0.356427],[1,-2,-2,0],[9E+09,9E+09,9E+09,9E+09,9E+09,9E+09]],s50,z10,a1\WObj:=grinder5;
    MoveL [[-86.18,-114.85,-238.02],[0.633686,0.629488,-0.251635,0.372647],[1,-2,-1,0],[9E+09,9E+09,9E+09,9E+09,9E+09,9E+09]],s50,z10,a1\WObj:=grinder5;
    MoveL [[-92.11,-123.97,-237.99],[0.572956,0.555375,-0.367831,0.477473],[1,-2,-1,0],[9E+09,9E+09,9E+09,9E+09,9E+09,9E+09]],s50,z10,a1\WObj:=grinder5;
    MoveL [[-92.10,-133.82,-237.96],[0.598604,0.518542,-0.324425,0.517239],[0,-2,-1,0],[9E+09,9E+09,9E+09,9E+09,9E+09,9E+09]],s50,z10,a1\WObj:=grinder5;
    MoveL [[-91.90,-116.15,-238.06],[0.570336,0.445227,-0.35666,0.591002],[1,-2,-1,0],[9E+09,9E+09,9E+09,9E+09,9E+09,9E+09]],s50,z10,a1\WObj:=grinder5;
    MoveL [[-95.09,-126.85,-238.08],[0.311286,0.305334,-0.455592,0.776085],[0,-2,0,0],[9E+09,9E+09,9E+09,9E+09,9E+09,9E+09]],s50,z10,a1\WObj:=grinder5;
    MoveL [[-100.35,-134.75,-238.08],[0.142001,0.101439,-0.534408,0.827015],[0,-2,0,0],[9E+09,9E+09,9E+09,9E+09,9E+09,9E+09]],s30,z10,a1\WObj:=grinder5;
    MoveL [[-91.41,-127.76,-238.13],[0.485957,0.437887,-0.41045,0.635321],[0,-2,-1,0],[9E+09,9E+09,9E+09,9E+09,9E+09,9E+09]],s50,z10,a1\WObj:=grinder5;
    MoveL [[-91.42,-129.94,-246.43],[0.524314,0.534591,-0.399458,0.528906],[1,-2,-1,0],[9E+09,9E+09,9E+09,9E+09,9E+09,9E+09]],s50,z10,a1\WObj:=grinder5;
    MoveL [[-91.90,-116.15,-238.06],[0.570336,0.445227,-0.35666,0.591002],[1,-2,-1,0],[9E+09,9E+09,9E+09,9E+09,9E+09,9E+09]],s100,z10,a1\WObj:=grinder5;
    MoveL [[-95.09,-126.85,-238.08],[0.311286,0.305334,-0.455592,0.776085],[0,-2,0,0],[9E+09,9E+09,9E+09,9E+09,9E+09,9E+09]],s50,z10,a1\WObj:=grinder5;
    MoveL [[-99.49,-134.82,-238.14],[0.081055,0.0552765,-0.535881,0.838574],[0,-2,0,0],[9E+09,9E+09,9E+09,9E+09,9E+09,9E+09]],s50,z10,a1\WObj:=grinder5;
    MoveL [[-91.41,-127.76,-238.13],[0.485957,0.437887,-0.41045,0.635321],[0,-2,-1,0],[9E+09,9E+09,9E+09,9E+09,9E+09,9E+09]],s50,z10,a1\WObj:=grinder5;
    MoveL [[-91.42,-129.94,-246.43],[0.524314,0.534591,-0.399458,0.528906],[1,-2,-1,0],[9E+09,9E+09,9E+09,9E+09,9E+09,9E+09]],s100,z10,a1\WObj:=grinder5;
    !
    S_WaxRed;
    !
    MoveL [[-91.44,-100.78,-246.46],[0.524298,0.53459,-0.399492,0.528896],[1,-2,-1,0],[9E+09,9E+09,9E+09,9E+09,9E+09,9E+09]],s50,z10,a1\WObj:=grinder5;
    MoveL [[-83.95,-100.83,-246.49],[0.664722,0.596991,0.0152785,0.448901],[0,-2,-1,0],[9E+09,9E+09,9E+09,9E+09,9E+09,9E+09]],s100,z10,a1\WObj:=grinder5;
    MoveL [[-83.97,-100.84,-246.51],[0.765263,0.567759,0.185184,0.240271],[0,-2,-2,0],[9E+09,9E+09,9E+09,9E+09,9E+09,9E+09]],s50,z10,a1\WObj:=grinder5;
    MoveL [[-83.98,-79.19,-246.54],[0.648385,0.549362,0.266272,0.45486],[0,-2,-1,0],[9E+09,9E+09,9E+09,9E+09,9E+09,9E+09]],s50,z10,a1\WObj:=grinder5;
    MoveL [[-85.74,-79.18,-246.54],[0.496433,0.601718,0.103124,0.617135],[0,-2,-1,0],[9E+09,9E+09,9E+09,9E+09,9E+09,9E+09]],s100,z10,a1\WObj:=grinder5;
    MoveL [[-83.98,-79.19,-246.54],[0.648385,0.549362,0.266272,0.45486],[0,-2,-1,0],[9E+09,9E+09,9E+09,9E+09,9E+09,9E+09]],s50,z10,a1\WObj:=grinder5;
    MoveL [[-83.98,-79.18,-246.54],[0.608099,0.491585,0.345913,0.518559],[0,-3,-1,0],[9E+09,9E+09,9E+09,9E+09,9E+09,9E+09]],s50,z10,a1\WObj:=grinder5;
    MoveL [[-83.98,-79.17,-246.54],[0.527365,0.536143,0.271775,0.600479],[0,-3,-1,0],[9E+09,9E+09,9E+09,9E+09,9E+09,9E+09]],s100,z10,a1\WObj:=grinder5;
    MoveL [[-84.00,-94.92,-246.58],[0.578796,0.670028,0.130309,0.446181],[0,-2,-1,0],[9E+09,9E+09,9E+09,9E+09,9E+09,9E+09]],s100,z10,a1\WObj:=grinder5;
    MoveL [[-84.00,-94.92,-246.58],[0.490809,0.682511,0.00981586,0.541469],[0,-2,-1,0],[9E+09,9E+09,9E+09,9E+09,9E+09,9E+09]],s100,z10,a1\WObj:=grinder5;
    MoveL [[-84.00,-94.92,-246.58],[0.622873,0.65242,0.200668,0.382243],[0,-2,-2,0],[9E+09,9E+09,9E+09,9E+09,9E+09,9E+09]],s100,z10,a1\WObj:=grinder5;
    MoveL [[-84.00,-115.11,-246.59],[0.652871,0.727472,0.0394604,0.207333],[1,-2,-2,0],[9E+09,9E+09,9E+09,9E+09,9E+09,9E+09]],s100,z10,a1\WObj:=grinder5;
    MoveL [[-86.97,-100.39,-246.60],[0.42892,0.627672,-0.369874,0.534086],[1,-2,-1,0],[9E+09,9E+09,9E+09,9E+09,9E+09,9E+09]],s100,z10,a1\WObj:=grinder5;
    MoveL [[-137.83,-97.92,-367.80],[0.428908,0.627655,-0.369883,0.53411],[1,-2,-1,0],[9E+09,9E+09,9E+09,9E+09,9E+09,9E+09]],s100,z50,a3\WObj:=grinder5;
    !
    MoveL [[-130.29,-113.64,-295.68],[0.127906,0.163224,-0.666189,0.716373],[1,-2,0,0],[9E+09,9E+09,9E+09,9E+09,9E+09,9E+09]],s300,z50,a3\WObj:=grinder5;
    MoveL [[-99.47,-113.63,-295.68],[0.0652067,0.104766,-0.677838,0.724781],[1,-2,0,0],[9E+09,9E+09,9E+09,9E+09,9E+09,9E+09]],s100,z10,a3\WObj:=grinder5;
    MoveL [[-99.55,-86.62,-295.73],[0.0199483,0.0622105,-0.683118,0.72738],[1,-2,0,0],[9E+09,9E+09,9E+09,9E+09,9E+09,9E+09]],s100,z10,a3\WObj:=grinder5;
    MoveL [[-99.52,-109.85,-295.71],[0.134888,0.169633,-0.66462,0.715059],[1,-2,0,0],[9E+09,9E+09,9E+09,9E+09,9E+09,9E+09]],s100,z10,a3\WObj:=grinder5;
    !
    MoveL [[-138.04,-108.52,-252.12],[0.562042,0.303144,0.660634,-0.394683],[0,-2,1,0],[9E+09,9E+09,9E+09,9E+09,9E+09,9E+09]],s300,z50,a3\WObj:=grinder5;
    MoveL [[-116.84,-111.20,-372.83],[0.562011,0.30312,0.660657,-0.394708],[0,-2,1,0],[9E+09,9E+09,9E+09,9E+09,9E+09,9E+09]],s100,z10,a1\WObj:=grinder5;
    MoveL [[-116.80,-89.13,-372.81],[0.457714,0.443069,0.537655,-0.552372],[1,-1,1,0],[9E+09,9E+09,9E+09,9E+09,9E+09,9E+09]],s100,z10,a1\WObj:=grinder5;
    MoveL [[-119.60,-116.77,-372.78],[0.457737,0.442981,0.537686,-0.552393],[1,-1,1,0],[9E+09,9E+09,9E+09,9E+09,9E+09,9E+09]],s100,z10,a1\WObj:=grinder5;
    MoveL [[-108.19,-110.12,-372.78],[0.517769,0.501424,0.483652,-0.496558],[1,-1,1,0],[9E+09,9E+09,9E+09,9E+09,9E+09,9E+09]],s100,z10,a1\WObj:=grinder5;
    MoveL [[-108.21,-87.88,-372.78],[0.517752,0.501447,0.483643,-0.496562],[1,-1,1,0],[9E+09,9E+09,9E+09,9E+09,9E+09,9E+09]],s100,z10,a1\WObj:=grinder5;
    MoveL [[-104.52,-85.05,-346.34],[0.572481,0.511687,0.468389,-0.437097],[1,-2,1,0],[9E+09,9E+09,9E+09,9E+09,9E+09,9E+09]],s100,z10,a1\WObj:=grinder5;
    MoveL [[-104.49,-116.49,-321.50],[0.572519,0.511639,0.468389,-0.437104],[1,-2,1,0],[9E+09,9E+09,9E+09,9E+09,9E+09,9E+09]],s100,z10,a1\WObj:=grinder5;
    MoveL [[-104.50,-116.49,-321.50],[0.522584,0.458724,0.520326,-0.49572],[1,-2,1,0],[9E+09,9E+09,9E+09,9E+09,9E+09,9E+09]],s50,z10,a1\WObj:=grinder5;
    MoveL [[-101.55,-95.90,-321.54],[0.633432,0.578242,0.383202,-0.342864],[1,-2,1,0],[9E+09,9E+09,9E+09,9E+09,9E+09,9E+09]],s100,z10,a1\WObj:=grinder5;
    MoveL [[-105.64,-95.91,-321.57],[0.529263,0.465912,0.513969,-0.48851],[1,-2,1,0],[9E+09,9E+09,9E+09,9E+09,9E+09,9E+09]],s50,z10,a1\WObj:=grinder5;
    MoveL [[-103.34,-102.65,-321.54],[0.338655,0.677226,0.602957,-0.251238],[0,-1,1,0],[9E+09,9E+09,9E+09,9E+09,9E+09,9E+09]],s50,z10,a1\WObj:=grinder5;
    MoveL [[-112.27,-109.37,-321.57],[0.23656,0.439821,0.792934,-0.349073],[0,-1,0,0],[9E+09,9E+09,9E+09,9E+09,9E+09,9E+09]],s50,z10,a1\WObj:=grinder5;
    MoveL [[-113.57,-117.53,-321.52],[0.222254,0.433702,0.801348,-0.34691],[0,-1,0,0],[9E+09,9E+09,9E+09,9E+09,9E+09,9E+09]],s50,z10,a1\WObj:=grinder5;
    MoveL [[-98.07,-106.77,-321.49],[0.728058,0.453035,0.441211,-0.264622],[0,-2,1,0],[9E+09,9E+09,9E+09,9E+09,9E+09,9E+09]],s100,z10,a1\WObj:=grinder5;
    MoveL [[-93.45,-93.75,-321.52],[0.706645,0.55044,0.4434,-0.032642],[0,-2,2,0],[9E+09,9E+09,9E+09,9E+09,9E+09,9E+09]],s100,z10,a1\WObj:=grinder5;
    MoveL [[-93.44,-93.74,-321.51],[0.72214,0.356795,0.577412,-0.13344],[0,-2,2,0],[9E+09,9E+09,9E+09,9E+09,9E+09,9E+09]],s100,z10,a1\WObj:=grinder5;
    MoveL [[-93.44,-93.75,-321.52],[0.692874,0.423613,0.582946,-0.0255225],[0,-2,2,0],[9E+09,9E+09,9E+09,9E+09,9E+09,9E+09]],s100,z10,a1\WObj:=grinder5;
    MoveL [[-99.40,-93.75,-321.56],[0.530754,0.614712,0.547394,-0.201965],[1,-1,1,0],[9E+09,9E+09,9E+09,9E+09,9E+09,9E+09]],s100,z10,a1\WObj:=grinder5;
    MoveL [[-95.99,-93.75,-321.49],[0.561019,0.714049,0.40934,-0.0885042],[1,-1,1,0],[9E+09,9E+09,9E+09,9E+09,9E+09,9E+09]],s100,z10,a1\WObj:=grinder5;
    MoveL [[-101.49,-122.16,-321.48],[0.633478,0.578183,0.383227,-0.342853],[1,-2,1,0],[9E+09,9E+09,9E+09,9E+09,9E+09,9E+09]],s100,z10,a1\WObj:=grinder5;
    MoveL [[-107.58,-116.52,-321.53],[0.536906,0.473777,0.506668,-0.480161],[1,-2,1,0],[9E+09,9E+09,9E+09,9E+09,9E+09,9E+09]],s100,z10,a1\WObj:=grinder5;
    MoveL [[-109.84,-84.97,-432.55],[0.558057,0.418648,0.559149,-0.447949],[1,-2,1,0],[9E+09,9E+09,9E+09,9E+09,9E+09,9E+09]],s100,z10,a1\WObj:=grinder5;
    MoveL [[-111.02,-112.48,-371.94],[0.526425,0.456069,0.532894,-0.480523],[1,-2,1,0],[9E+09,9E+09,9E+09,9E+09,9E+09,9E+09]],s100,z10,a1\WObj:=grinder5;
    MoveL [[-111.07,-82.54,-371.97],[0.52639,0.456121,0.532884,-0.480523],[1,-2,1,0],[9E+09,9E+09,9E+09,9E+09,9E+09,9E+09]],s100,z10,a1\WObj:=grinder5;
    MoveL [[-157.04,-82.49,-267.45],[0.557934,0.418672,0.559221,-0.447989],[1,-2,1,0],[9E+09,9E+09,9E+09,9E+09,9E+09,9E+09]],s200,z50,a3\WObj:=grinder5;
    !
    MoveL [[-167.13,-82.42,-310.63],[0.173933,0.548168,0.798071,0.179839],[0,0,0,0],[9E+09,9E+09,9E+09,9E+09,9E+09,9E+09]],s200,z50,a3\WObj:=grinder5;
    !
    MoveL [[-102.15,-82.43,-310.63],[0.231377,0.496863,0.801553,0.238966],[0,0,0,0],[9E+09,9E+09,9E+09,9E+09,9E+09,9E+09]],s200,z10,a3\WObj:=grinder5;
    MoveL [[-102.72,-103.27,-340.82],[0.00732049,0.569943,0.810082,-0.137397],[0,-1,0,0],[9E+09,9E+09,9E+09,9E+09,9E+09,9E+09]],s100,z10,a3\WObj:=grinder5;
    MoveL [[-101.57,-146.42,-274.71],[0.352099,0.562412,0.74446,0.0741519],[0,-1,0,0],[9E+09,9E+09,9E+09,9E+09,9E+09,9E+09]],s100,z10,a3\WObj:=grinder5;
    MoveL [[-113.12,-163.06,-303.47],[0.119365,0.679047,0.699979,-0.186218],[0,-1,0,0],[9E+09,9E+09,9E+09,9E+09,9E+09,9E+09]],s100,z10,a3\WObj:=grinder5;
    MoveL [[-133.87,-180.49,-294.67],[0.425329,0.662274,0.603249,0.128758],[0,-1,1,0],[9E+09,9E+09,9E+09,9E+09,9E+09,9E+09]],s100,z10,a3\WObj:=grinder5;
    MoveL [[-123.61,-176.49,-284.60],[0.243067,0.688067,0.641005,-0.237896],[0,-1,1,0],[9E+09,9E+09,9E+09,9E+09,9E+09,9E+09]],s50,z10,a3\WObj:=grinder5;
    MoveL [[-141.64,-184.90,-346.59],[0.370112,0.723433,0.543518,0.210358],[0,-1,1,0],[9E+09,9E+09,9E+09,9E+09,9E+09,9E+09]],s100,z10,a3\WObj:=grinder5;
    !
    MoveL [[-165.96,-184.78,-346.64],[0.260824,-0.399891,0.83186,-0.282962],[0,0,-2,0],[9E+09,9E+09,9E+09,9E+09,9E+09,9E+09]],s300,z100,a3\WObj:=grinder5;
    !
    S_WaxRed;
    !
    MoveL [[-142.69,-230.51,-309.79],[0.464741,-0.554994,0.465788,-0.508959],[0,1,-3,0],[9E+09,9E+09,9E+09,9E+09,9E+09,9E+09]],s300,z50,a1\WObj:=grinder5;
    MoveL [[-107.99,-219.53,-309.83],[0.550977,-0.441444,0.369398,-0.604233],[0,1,-3,0],[9E+09,9E+09,9E+09,9E+09,9E+09,9E+09]],s300,z10,a1\WObj:=grinder5;
    MoveL [[-112.95,-116.96,-302.65],[0.550117,-0.442361,0.370555,-0.603637],[0,1,-3,0],[9E+09,9E+09,9E+09,9E+09,9E+09,9E+09]],s50,z10,a1\WObj:=grinder5;
    MoveL [[-109.05,-116.88,-309.87],[0.504845,-0.493516,0.427051,-0.564979],[0,1,-3,0],[9E+09,9E+09,9E+09,9E+09,9E+09,9E+09]],s50,z10,a1\WObj:=grinder5;
    MoveL [[-108.67,-200.69,-309.97],[0.49411,-0.504258,0.43901,-0.555742],[0,1,-3,0],[9E+09,9E+09,9E+09,9E+09,9E+09,9E+09]],s50,z10,a1\WObj:=grinder5;
    MoveL [[-99.69,-116.38,-309.89],[0.385849,-0.605967,0.603271,-0.346394],[0,0,-3,0],[9E+09,9E+09,9E+09,9E+09,9E+09,9E+09]],s50,z10,a1\WObj:=grinder5;
    MoveL [[-99.70,-206.89,-309.89],[0.385848,-0.605953,0.603289,-0.346389],[0,0,-3,0],[9E+09,9E+09,9E+09,9E+09,9E+09,9E+09]],s100,z10,a1\WObj:=grinder5;
    MoveL [[-99.71,-206.89,-309.89],[0.253123,-0.680742,0.650557,-0.222021],[0,0,-2,0],[9E+09,9E+09,9E+09,9E+09,9E+09,9E+09]],s100,z10,a1\WObj:=grinder5;
    MoveL [[-98.42,-159.16,-309.90],[0.253109,-0.680769,0.650534,-0.222024],[0,0,-2,0],[9E+09,9E+09,9E+09,9E+09,9E+09,9E+09]],s100,z10,a1\WObj:=grinder5;
    MoveL [[-98.45,-107.54,-309.93],[0.253065,-0.680811,0.650507,-0.222027],[0,0,-2,0],[9E+09,9E+09,9E+09,9E+09,9E+09,9E+09]],s100,z10,a1\WObj:=grinder5;
    MoveL [[-88.82,-195.18,-309.92],[0.189565,-0.741163,0.618366,-0.179907],[0,0,-2,0],[9E+09,9E+09,9E+09,9E+09,9E+09,9E+09]],s50,z10,a1\WObj:=grinder5;
    MoveL [[-94.58,-163.58,-309.97],[0.198652,-0.707811,0.656301,-0.169732],[0,0,-2,0],[9E+09,9E+09,9E+09,9E+09,9E+09,9E+09]],s50,z10,a1\WObj:=grinder5;
    MoveL [[-100.68,-106.79,-309.98],[0.209413,-0.663082,0.701457,-0.15629],[0,0,-2,0],[9E+09,9E+09,9E+09,9E+09,9E+09,9E+09]],s50,z10,a1\WObj:=grinder5;
    MoveL [[-99.69,-116.38,-309.89],[0.151874,-0.672032,0.719099,-0.0905728],[0,0,-2,0],[9E+09,9E+09,9E+09,9E+09,9E+09,9E+09]],s50,z10,a1\WObj:=grinder5;
    MoveL [[-89.48,-163.49,-309.95],[0.142443,-0.737743,0.651523,-0.104704],[0,0,-2,0],[9E+09,9E+09,9E+09,9E+09,9E+09,9E+09]],s50,z10,a1\WObj:=grinder5;
    MoveL [[-83.81,-193.78,-309.98],[0.139517,-0.755367,0.631006,-0.108563],[0,0,-2,0],[9E+09,9E+09,9E+09,9E+09,9E+09,9E+09]],s50,z10,a1\WObj:=grinder5;
    MoveL [[-87.55,-191.91,-309.95],[0.0537133,-0.76106,0.638556,0.100735],[0,0,-2,0],[9E+09,9E+09,9E+09,9E+09,9E+09,9E+09]],s50,z10,a1\WObj:=grinder5;
    MoveL [[-99.28,-151.33,-297.83],[0.070539,-0.699433,0.69733,0.139819],[0,0,-2,0],[9E+09,9E+09,9E+09,9E+09,9E+09,9E+09]],s50,z10,a1\WObj:=grinder5;
    MoveL [[-103.67,-89.17,-279.19],[0.089941,-0.611006,0.760114,0.202014],[0,0,-2,0],[9E+09,9E+09,9E+09,9E+09,9E+09,9E+09]],s50,z10,a1\WObj:=grinder5;
    MoveL [[-87.52,-193.71,-309.93],[0.0138757,-0.768292,0.616875,0.170296],[0,0,-2,0],[9E+09,9E+09,9E+09,9E+09,9E+09,9E+09]],s50,z10,a1\WObj:=grinder5;
    MoveL [[-97.04,-139.43,-294.00],[0.0584059,-0.70614,0.681743,0.182157],[0,0,-2,0],[9E+09,9E+09,9E+09,9E+09,9E+09,9E+09]],s50,z10,a1\WObj:=grinder5;
    MoveL [[-102.34,-89.18,-279.22],[0.096429,-0.635471,0.739784,0.198992],[0,0,-2,0],[9E+09,9E+09,9E+09,9E+09,9E+09,9E+09]],s50,z10,a1\WObj:=grinder5;
    MoveL [[-87.52,-193.71,-309.93],[0.0138757,-0.768292,0.616875,0.170296],[0,0,-2,0],[9E+09,9E+09,9E+09,9E+09,9E+09,9E+09]],s50,z10,a1\WObj:=grinder5;
    !
    MoveJ [[-392.60,-67.92,-310.53],[0.0014141,-0.77267,0.634794,-0.0040009],[0,0,-2,0],[9E+09,9E+09,9E+09,9E+09,9E+09,9E+09]],s500,z50,a3\WObj:=grinder5;
    MoveJ [[-222.54,-87.69,-310.63],[0.181653,-0.509374,-0.496869,-0.678721],[0,0,0,0],[9E+09,9E+09,9E+09,9E+09,9E+09,9E+09]],s300,z50,a3\WObj:=grinder5;
    MoveL [[-120.61,-87.69,-310.64],[0.181628,-0.509356,-0.49688,-0.678732],[0,0,0,0],[9E+09,9E+09,9E+09,9E+09,9E+09,9E+09]],s500,z50,a3\WObj:=grinder5;
    !
    S_WaxRed;
    !
    MoveL [[-96.27,-87.72,-310.60],[0.181607,-0.509343,-0.49688,-0.678748],[0,0,0,0],[9E+09,9E+09,9E+09,9E+09,9E+09,9E+09]],s200,z10,a3\WObj:=grinder5;
    MoveL [[-101.54,-87.67,-310.65],[0.290316,-0.456258,-0.635311,-0.551294],[0,0,0,0],[9E+09,9E+09,9E+09,9E+09,9E+09,9E+09]],s100,z10,a3\WObj:=grinder5;
    MoveL [[-99.70,-87.66,-310.64],[0.26141,-0.498765,-0.719505,-0.406462],[0,0,0,0],[9E+09,9E+09,9E+09,9E+09,9E+09,9E+09]],s100,z10,a3\WObj:=grinder5;
    MoveL [[-104.60,-87.67,-310.66],[0.322999,-0.460622,-0.76314,-0.317989],[0,0,0,0],[9E+09,9E+09,9E+09,9E+09,9E+09,9E+09]],s50,z10,a3\WObj:=grinder5;
    MoveL [[-101.09,-135.47,-425.09],[0.320687,-0.526386,-0.713368,-0.33344],[0,0,0,0],[9E+09,9E+09,9E+09,9E+09,9E+09,9E+09]],s50,z10,a3\WObj:=grinder5;
    MoveL [[-100.23,-163.59,-433.06],[0.348769,-0.547536,-0.703247,-0.289841],[0,0,0,0],[9E+09,9E+09,9E+09,9E+09,9E+09,9E+09]],s100,z10,a3\WObj:=grinder5;
    MoveL [[-162.25,-153.02,-416.38],[0.344149,-0.772539,-0.473149,-0.246726],[0,0,0,0],[9E+09,9E+09,9E+09,9E+09,9E+09,9E+09]],s100,z10,a3\WObj:=grinder5;
    MoveL [[-124.66,-130.01,-372.31],[0.235302,-0.696877,-0.614926,-0.284363],[0,0,0,0],[9E+09,9E+09,9E+09,9E+09,9E+09,9E+09]],s100,z10,a3\WObj:=grinder5;
    MoveL [[-103.92,-81.75,-310.65],[0.21177,-0.548793,-0.77005,-0.246987],[0,0,0,0],[9E+09,9E+09,9E+09,9E+09,9E+09,9E+09]],s100,z10,a3\WObj:=grinder5;
    MoveL [[-113.21,-139.17,-310.71],[0.244017,-0.650429,-0.686376,-0.215142],[0,0,0,0],[9E+09,9E+09,9E+09,9E+09,9E+09,9E+09]],s100,z10,a3\WObj:=grinder5;
    MoveL [[-104.76,-117.27,-310.70],[0.164673,-0.677816,-0.605819,-0.382663],[0,0,0,0],[9E+09,9E+09,9E+09,9E+09,9E+09,9E+09]],s100,z10,a3\WObj:=grinder5;
    MoveL [[-99.70,-87.66,-310.64],[0.23233,-0.512954,-0.694977,-0.447111],[0,0,0,0],[9E+09,9E+09,9E+09,9E+09,9E+09,9E+09]],s100,z10,a3\WObj:=grinder5;
    MoveL [[-101.55,-87.67,-310.67],[0.28663,-0.45859,-0.630855,-0.556382],[0,0,0,0],[9E+09,9E+09,9E+09,9E+09,9E+09,9E+09]],s100,z10,a3\WObj:=grinder5;
    MoveL [[-104.49,-101.74,-383.73],[0.174276,-0.556189,-0.695755,-0.419771],[0,0,0,0],[9E+09,9E+09,9E+09,9E+09,9E+09,9E+09]],s100,z10,a3\WObj:=grinder5;
    MoveL [[-109.76,-133.14,-417.97],[0.176907,-0.668271,-0.628533,-0.35646],[0,0,0,0],[9E+09,9E+09,9E+09,9E+09,9E+09,9E+09]],s100,z10,a3\WObj:=grinder5;
    MoveL [[-101.78,-72.11,-331.58],[0.21533,-0.733845,-0.550578,-0.334617],[0,0,0,0],[9E+09,9E+09,9E+09,9E+09,9E+09,9E+09]],s100,z10,a1\WObj:=grinder5;
    MoveL [[-101.77,-72.12,-331.58],[0.418112,-0.828737,-0.285796,-0.238114],[0,0,1,0],[9E+09,9E+09,9E+09,9E+09,9E+09,9E+09]],s100,z10,a1\WObj:=grinder5;
    MoveL [[-101.78,-72.11,-331.58],[0.21533,-0.733845,-0.550578,-0.334617],[0,0,0,0],[9E+09,9E+09,9E+09,9E+09,9E+09,9E+09]],s100,z10,a1\WObj:=grinder5;
    MoveL [[-109.76,-133.14,-417.97],[0.176907,-0.668271,-0.628533,-0.35646],[0,0,0,0],[9E+09,9E+09,9E+09,9E+09,9E+09,9E+09]],s100,z10,a3\WObj:=grinder5;
    MoveL [[-104.49,-101.74,-383.73],[0.174276,-0.556189,-0.695755,-0.419771],[0,0,0,0],[9E+09,9E+09,9E+09,9E+09,9E+09,9E+09]],s100,z10,a3\WObj:=grinder5;
    MoveL [[-103.01,-82.61,-335.50],[0.147216,-0.456051,-0.780236,-0.401966],[0,0,0,0],[9E+09,9E+09,9E+09,9E+09,9E+09,9E+09]],s50,z10,a3\WObj:=grinder5;
    !
    MoveL [[-238.29,-25.07,-251.47],[0.115726,-0.45663,-0.76482,-0.439485],[0,0,0,0],[9E+09,9E+09,9E+09,9E+09,9E+09,9E+09]],s500,z50,a1\WObj:=grinder5;
    MoveL [[-426.53,-72.18,-331.58],[0.0960727,-0.205663,0.972343,-0.0549636],[0,0,-1,0],[9E+09,9E+09,9E+09,9E+09,9E+09,9E+09]],s500,z50,a1\WObj:=grinder5;
    !!
    S_Grinder5 "Stop";
ENDPROC

!******************************
PROC R_Polish6()
    P_OffsetCalculation 6;
    !
    !! Warning! Engine starting
    S_Grinder6 "Start";
    !!
    S_WaxWhite;
    !
    MoveL [[-399.04,-244.47,-197.44],[5.64595E-06,0.0289272,-0.999582,-2.41436E-05],[1,0,0,0],[9E+09,9E+09,9E+09,9E+09,9E+09,9E+09]],s800,z50,tool1\WObj:=grinder6;
    !
    T_RotateX;
    !
    MoveL [[-392.96,32.21,-249.00],[0.404593,-0.145026,0.747474,-0.506512],[1,-1,0,0],[9E+09,9E+09,9E+09,9E+09,9E+09,9E+09]],s800,z50,b1\WObj:=grinder6;
    !
    MoveL [[-157.25,121.25,-286.06],[0.284811,-0.065527,0.800792,-0.522802],[1,-1,0,0],[9E+09,9E+09,9E+09,9E+09,9E+09,9E+09]],s500,z50,b1\WObj:=grinder6;
    MoveL [[-124.27,121.86,-308.31],[0.280462,0.00207546,0.813271,-0.50983],[1,-1,0,0],[9E+09,9E+09,9E+09,9E+09,9E+09,9E+09]],s100,z5,b1\WObj:=grinder6;
    MoveL [[-85.95,44.72,-330.52],[0.28042,0.00205382,0.813294,-0.509817],[1,-1,0,0],[9E+09,9E+09,9E+09,9E+09,9E+09,9E+09]],s100,z5,b1\WObj:=grinder6;
    MoveL [[-85.34,36.35,-335.18],[0.183601,-0.145024,0.80023,-0.552169],[1,-1,0,0],[9E+09,9E+09,9E+09,9E+09,9E+09,9E+09]],s50,z5,b1\WObj:=grinder6;
    MoveL [[-68.88,25.95,-337.24],[0.353486,-0.25757,0.720542,-0.538075],[1,-2,0,0],[9E+09,9E+09,9E+09,9E+09,9E+09,9E+09]],s50,z5,b1\WObj:=grinder6;
    MoveL [[-63.39,28.10,-337.15],[0.388543,-0.21161,0.642044,-0.626127],[1,-2,0,0],[9E+09,9E+09,9E+09,9E+09,9E+09,9E+09]],s50,z5,b1\WObj:=grinder6;
    MoveL [[-87.98,38.18,-327.01],[0.168275,-0.11955,0.784663,-0.584547],[1,-1,0,0],[9E+09,9E+09,9E+09,9E+09,9E+09,9E+09]],s50,z5,b1\WObj:=grinder6;
    MoveL [[-118.98,111.03,-305.26],[0.111085,-0.10398,0.868818,-0.471173],[1,-1,0,0],[9E+09,9E+09,9E+09,9E+09,9E+09,9E+09]],s100,z5,b1\WObj:=grinder6;
    MoveL [[-120.33,119.98,-302.93],[0.124759,-0.0870916,0.792906,-0.590042],[1,-1,0,0],[9E+09,9E+09,9E+09,9E+09,9E+09,9E+09]],s50,z5,b1\WObj:=grinder6;
    MoveL [[-81.48,36.13,-297.07],[0.235099,-0.0448323,0.783953,-0.572831],[1,-1,0,0],[9E+09,9E+09,9E+09,9E+09,9E+09,9E+09]],s100,z5,b1\WObj:=grinder6;
    MoveL [[-120.12,120.07,-302.99],[0.124678,-0.087065,0.792953,-0.590001],[1,-1,0,0],[9E+09,9E+09,9E+09,9E+09,9E+09,9E+09]],s100,z5,b1\WObj:=grinder6;
    MoveL [[-81.62,37.01,-297.07],[0.235098,-0.0448319,0.783951,-0.572835],[1,-1,0,0],[9E+09,9E+09,9E+09,9E+09,9E+09,9E+09]],s100,z5,b1\WObj:=grinder6;
    MoveL [[-51.69,36.23,-297.08],[0.443677,-0.202146,0.687726,-0.537885],[1,-2,0,0],[9E+09,9E+09,9E+09,9E+09,9E+09,9E+09]],s50,z5,b1\WObj:=grinder6;
    MoveL [[-55.53,31.70,-297.04],[0.166839,-0.480285,0.532111,-0.677014],[1,-2,0,0],[9E+09,9E+09,9E+09,9E+09,9E+09,9E+09]],s50,z5,b1\WObj:=grinder6;
    MoveL [[-50.79,35.51,-297.16],[0.443571,-0.202117,0.687823,-0.53786],[1,-2,0,0],[9E+09,9E+09,9E+09,9E+09,9E+09,9E+09]],s50,z5,b1\WObj:=grinder6;
    MoveL [[-55.28,32.47,-297.15],[0.166761,-0.480229,0.532325,-0.676905],[1,-2,0,0],[9E+09,9E+09,9E+09,9E+09,9E+09,9E+09]],s50,z5,b1\WObj:=grinder6;
    MoveL [[-81.31,35.17,-297.07],[0.235169,-0.0448527,0.783906,-0.572866],[1,-1,0,0],[9E+09,9E+09,9E+09,9E+09,9E+09,9E+09]],s50,z5,b1\WObj:=grinder6;
    MoveL [[-123.70,123.61,-297.10],[0.234952,-0.0449073,0.784058,-0.572742],[1,-1,0,0],[9E+09,9E+09,9E+09,9E+09,9E+09,9E+09]],s100,z5,b1\WObj:=grinder6;
    !
    MoveL [[-220.52,123.59,-297.16],[0.234975,-0.0448646,0.784037,-0.572765],[1,-1,0,0],[9E+09,9E+09,9E+09,9E+09,9E+09,9E+09]],s500,z50,b1\WObj:=grinder6;
    MoveL [[-650.35,123.58,-297.11],[0.0167125,-0.161637,0.986638,0.0118163],[1,0,0,0],[9E+09,9E+09,9E+09,9E+09,9E+09,9E+09]],s500,z50,b1\WObj:=grinder6;
    !
    T_RotateZ;
    !
    S_WaxWhite;
    !
    MoveL [[-231.03,55.91,-359.08],[0.0721434,-0.161913,0.983993,-0.018384],[1,-1,0,0],[9E+09,9E+09,9E+09,9E+09,9E+09,9E+09]],s500,z50,a1\WObj:=grinder6;
    !
    MoveL [[-205.08,52.26,-359.09],[0.072128,-0.161956,0.983986,-0.0183932],[1,-1,0,0],[9E+09,9E+09,9E+09,9E+09,9E+09,9E+09]],s100,z5,a1\WObj:=grinder6;
    MoveL [[-207.09,45.10,-332.21],[0.0721477,-0.162007,0.983975,-0.0184639],[1,-1,0,0],[9E+09,9E+09,9E+09,9E+09,9E+09,9E+09]],s50,z5,a1\WObj:=grinder6;
    MoveL [[-203.20,59.91,-332.17],[0.0722672,-0.162171,0.983934,-0.0187628],[1,-1,0,0],[9E+09,9E+09,9E+09,9E+09,9E+09,9E+09]],s50,z5,a1\WObj:=grinder6;
    MoveL [[-210.45,57.17,-332.26],[0.0941246,-0.125477,0.911989,-0.379041],[1,-1,0,0],[9E+09,9E+09,9E+09,9E+09,9E+09,9E+09]],s100,z5,a1\WObj:=grinder6;
    MoveL [[-193.67,17.61,-305.67],[0.0408299,-0.250446,0.885803,-0.38854],[1,-1,0,0],[9E+09,9E+09,9E+09,9E+09,9E+09,9E+09]],s50,z5,a1\WObj:=grinder6;
    MoveL [[-209.63,53.02,-332.20],[0.0941939,-0.125464,0.911945,-0.379134],[1,-1,0,0],[9E+09,9E+09,9E+09,9E+09,9E+09,9E+09]],s50,z5,a1\WObj:=grinder6;
    MoveL [[-200.74,43.92,-332.12],[0.115778,-0.232185,0.904316,0.338966],[1,0,-1,0],[9E+09,9E+09,9E+09,9E+09,9E+09,9E+09]],s100,z5,a1\WObj:=grinder6;
    MoveL [[-181.94,36.55,-376.57],[0.162274,-0.356736,0.862748,0.319487],[1,0,-1,0],[9E+09,9E+09,9E+09,9E+09,9E+09,9E+09]],s100,z5,a1\WObj:=grinder6;
    MoveL [[-204.61,48.60,-332.48],[0.0721371,-0.161914,0.983995,-0.0182788],[1,-1,0,0],[9E+09,9E+09,9E+09,9E+09,9E+09,9E+09]],s100,z5,a1\WObj:=grinder6;
    !
    MoveL [[-302.86,50.09,-332.54],[0.0721586,-0.162041,0.983968,-0.0185307],[1,-1,0,0],[9E+09,9E+09,9E+09,9E+09,9E+09,9E+09]],s500,z50,a1\WObj:=grinder6;
    MoveL [[-151.69,72.74,-233.96],[0.513887,-0.478241,0.470612,-0.534537],[1,-2,0,0],[9E+09,9E+09,9E+09,9E+09,9E+09,9E+09]],s200,z50,a1\WObj:=grinder6;
    !
    MoveL [[-83.96,72.77,-233.94],[0.513894,-0.478286,0.470529,-0.534563],[1,-2,0,0],[9E+09,9E+09,9E+09,9E+09,9E+09,9E+09]],s100,z5,a1\WObj:=grinder6;
    MoveL [[-80.86,-39.39,-227.25],[0.484929,-0.502451,0.444601,-0.560997],[1,-2,0,0],[9E+09,9E+09,9E+09,9E+09,9E+09,9E+09]],s50,z5,a1\WObj:=grinder6;
    MoveL [[-81.75,-39.39,-227.24],[0.431698,-0.548874,0.499015,-0.513185],[1,-2,0,0],[9E+09,9E+09,9E+09,9E+09,9E+09,9E+09]],s50,z5,a1\WObj:=grinder6;
    MoveL [[-78.06,77.54,-227.28],[0.431706,-0.548889,0.499014,-0.513163],[1,-2,0,0],[9E+09,9E+09,9E+09,9E+09,9E+09,9E+09]],s50,z5,a1\WObj:=grinder6;
    MoveL [[-78.32,-34.47,-238.87],[0.291438,-0.672852,0.540952,-0.411953],[1,-1,-1,0],[9E+09,9E+09,9E+09,9E+09,9E+09,9E+09]],s100,z5,a1\WObj:=grinder6;
    MoveL [[-87.18,22.44,-259.76],[0.351321,-0.581593,0.638093,-0.36216],[1,-1,0,0],[9E+09,9E+09,9E+09,9E+09,9E+09,9E+09]],s100,z5,a1\WObj:=grinder6;
    MoveL [[-85.30,79.26,-258.10],[0.351356,-0.581659,0.637959,-0.362256],[1,-1,0,0],[9E+09,9E+09,9E+09,9E+09,9E+09,9E+09]],s100,z5,a1\WObj:=grinder6;
    MoveL [[-86.88,83.45,-274.23],[0.179915,-0.664631,0.707138,-0.160786],[1,-1,-1,0],[9E+09,9E+09,9E+09,9E+09,9E+09,9E+09]],s100,z5,a1\WObj:=grinder6;
    MoveL [[-76.29,27.20,-278.09],[0.166803,-0.717589,0.653349,-0.174291],[1,-1,-1,0],[9E+09,9E+09,9E+09,9E+09,9E+09,9E+09]],s100,z5,a1\WObj:=grinder6;
    MoveL [[-61.05,-30.81,-275.88],[0.144971,-0.782305,0.573949,-0.193816],[1,-1,-1,0],[9E+09,9E+09,9E+09,9E+09,9E+09,9E+09]],s100,z5,a1\WObj:=grinder6;
    MoveL [[-57.22,-31.56,-284.49],[0.0090848,0.816146,-0.577549,0.0161352],[1,-1,-2,0],[9E+09,9E+09,9E+09,9E+09,9E+09,9E+09]],s100,z5,a1\WObj:=grinder6;
    MoveL [[-74.53,25.84,-286.83],[0.00740655,0.754388,-0.656172,0.0168023],[1,-1,-1,0],[9E+09,9E+09,9E+09,9E+09,9E+09,9E+09]],s50,z5,a1\WObj:=grinder6;
    MoveL [[-91.08,88.44,-285.53],[0.00437251,0.62861,-0.777504,0.0178224],[1,-1,-1,0],[9E+09,9E+09,9E+09,9E+09,9E+09,9E+09]],s50,z5,a1\WObj:=grinder6;
    MoveL [[-74.08,25.80,-293.19],[0.00740705,0.75438,-0.656179,0.0168531],[1,-1,-1,0],[9E+09,9E+09,9E+09,9E+09,9E+09,9E+09]],s50,z5,a1\WObj:=grinder6;
    MoveL [[-57.12,-31.00,-297.93],[0.00902441,0.816143,-0.577558,0.0160312],[1,-1,-2,0],[9E+09,9E+09,9E+09,9E+09,9E+09,9E+09]],s50,z5,a1\WObj:=grinder6;
    !
    S_WaxWhite;
    !
    MoveL [[-152.71,90.14,-240.08],[0.00902574,0.81616,-0.577535,0.0159866],[1,-1,-2,0],[9E+09,9E+09,9E+09,9E+09,9E+09,9E+09]],s300,z50,a3\WObj:=grinder6;
    MoveL [[-147.94,90.21,-321.65],[0.275061,0.569914,0.740429,0.226505],[1,-1,1,0],[9E+09,9E+09,9E+09,9E+09,9E+09,9E+09]],s300,z50,a3\WObj:=grinder6;
    !
    MoveL [[-128.63,199.97,-336.57],[0.294643,0.499813,0.789438,0.2004],[1,-1,1,0],[9E+09,9E+09,9E+09,9E+09,9E+09,9E+09]],s300,z5,a1\WObj:=grinder6;
    MoveL [[-111.74,152.77,-323.90],[0.274876,0.570122,0.740339,0.2265],[1,-1,1,0],[9E+09,9E+09,9E+09,9E+09,9E+09,9E+09]],s100,z5,a1\WObj:=grinder6;
    MoveL [[-91.94,100.84,-302.47],[0.222055,0.711079,0.6062,0.278531],[1,-1,1,0],[9E+09,9E+09,9E+09,9E+09,9E+09,9E+09]],s100,z5,a1\WObj:=grinder6;
    MoveL [[-88.59,90.68,-302.50],[0.0929671,0.742498,0.644096,0.158725],[1,-1,1,0],[9E+09,9E+09,9E+09,9E+09,9E+09,9E+09]],s100,z5,a1\WObj:=grinder6;
    MoveL [[-105.95,147.61,-302.49],[0.112689,0.653183,0.734512,0.145413],[1,-1,1,0],[9E+09,9E+09,9E+09,9E+09,9E+09,9E+09]],s100,z5,a1\WObj:=grinder6;
    MoveL [[-128.75,202.13,-302.47],[0.132091,0.543293,0.819131,0.128095],[1,-1,1,0],[9E+09,9E+09,9E+09,9E+09,9E+09,9E+09]],s100,z5,a1\WObj:=grinder6;
    MoveL [[-129.13,203.62,-302.49],[0.0469764,0.557167,0.82907,0.000633477],[1,-1,1,0],[9E+09,9E+09,9E+09,9E+09,9E+09,9E+09]],s100,z5,a1\WObj:=grinder6;
    MoveL [[-108.64,152.46,-302.52],[0.0464809,0.642614,0.764758,0.00568494],[1,-1,1,0],[9E+09,9E+09,9E+09,9E+09,9E+09,9E+09]],s100,z5,a1\WObj:=grinder6;
    MoveL [[-90.73,88.04,-302.53],[0.0456018,0.720071,0.692319,0.0105764],[1,-1,1,0],[9E+09,9E+09,9E+09,9E+09,9E+09,9E+09]],s100,z5,a1\WObj:=grinder6;
    MoveL [[-109.61,152.42,-302.50],[0.0465447,0.64261,0.764757,0.00567732],[1,-1,1,0],[9E+09,9E+09,9E+09,9E+09,9E+09,9E+09]],s100,z5,a1\WObj:=grinder6;
    MoveL [[-129.32,201.69,-302.46],[0.0470206,0.557134,0.82909,0.000643207],[1,-1,1,0],[9E+09,9E+09,9E+09,9E+09,9E+09,9E+09]],s100,z5,a1\WObj:=grinder6;
    !
    MoveL [[-195.86,165.40,-287.73],[0.0628448,-0.55544,-0.80616,-0.194017],[1,0,0,0],[9E+09,9E+09,9E+09,9E+09,9E+09,9E+09]],s500,z50,a1\WObj:=grinder6;
    MoveL [[-195.84,91.74,-248.17],[0.325926,-0.420215,-0.557404,-0.637567],[0,1,0,0],[9E+09,9E+09,9E+09,9E+09,9E+09,9E+09]],s300,z50,a1\WObj:=grinder6;
    !
    MoveL [[-142.05,91.76,-200.46],[0.315297,-0.410854,-0.564392,-0.642844],[0,1,0,0],[9E+09,9E+09,9E+09,9E+09,9E+09,9E+09]],s300,z5,a1\WObj:=grinder6;
    MoveL [[-111.62,87.52,-225.51],[0.417271,-0.498532,-0.488719,-0.581811],[0,1,0,0],[9E+09,9E+09,9E+09,9E+09,9E+09,9E+09]],s100,z5,a1\WObj:=grinder6;
    MoveL [[-93.28,87.48,-273.28],[0.507391,-0.572212,-0.3997,-0.505339],[0,1,0,0],[9E+09,9E+09,9E+09,9E+09,9E+09,9E+09]],s100,z5,a1\WObj:=grinder6;
    MoveL [[-112.36,87.52,-251.31],[0.462704,-0.456933,-0.543111,-0.531176],[0,0,0,0],[9E+09,9E+09,9E+09,9E+09,9E+09,9E+09]],s100,z5,a1\WObj:=grinder6;
    MoveL [[-144.81,91.77,-230.59],[0.37676,-0.354686,-0.656958,-0.548321],[0,0,0,0],[9E+09,9E+09,9E+09,9E+09,9E+09,9E+09]],s100,z5,a1\WObj:=grinder6;
    MoveL [[-112.24,87.53,-251.33],[0.462718,-0.456963,-0.543114,-0.531135],[0,0,0,0],[9E+09,9E+09,9E+09,9E+09,9E+09,9E+09]],s100,z5,a1\WObj:=grinder6;
    MoveL [[-96.29,87.50,-277.93],[0.544751,-0.524537,-0.44814,-0.476737],[0,0,0,0],[9E+09,9E+09,9E+09,9E+09,9E+09,9E+09]],s100,z5,a1\WObj:=grinder6;
    MoveL [[-87.65,123.97,-277.95],[0.500795,-0.566293,-0.407086,-0.512638],[0,1,0,0],[9E+09,9E+09,9E+09,9E+09,9E+09,9E+09]],s100,z5,a1\WObj:=grinder6;
    MoveL [[-85.29,126.22,-277.89],[0.597198,-0.639881,-0.278828,-0.395173],[0,1,0,0],[9E+09,9E+09,9E+09,9E+09,9E+09,9E+09]],s50,z5,a1\WObj:=grinder6;
    MoveL [[-88.19,123.69,-277.90],[0.450185,-0.393726,-0.379305,-0.706003],[1,1,0,0],[9E+09,9E+09,9E+09,9E+09,9E+09,9E+09]],s50,z5,a1\WObj:=grinder6;
    MoveL [[-86.68,115.84,-277.94],[0.597193,-0.639917,-0.278867,-0.395095],[0,1,0,0],[9E+09,9E+09,9E+09,9E+09,9E+09,9E+09]],s50,z5,a1\WObj:=grinder6;
    MoveL [[-88.51,98.35,-278.01],[0.678448,-0.50572,-0.207932,-0.490632],[0,1,0,0],[9E+09,9E+09,9E+09,9E+09,9E+09,9E+09]],s50,z5,a1\WObj:=grinder6;
    MoveL [[-99.74,104.41,-277.93],[0.417334,-0.322772,-0.470245,-0.707475],[0,1,0,0],[9E+09,9E+09,9E+09,9E+09,9E+09,9E+09]],s100,z5,a1\WObj:=grinder6;
    MoveL [[-102.94,108.83,-277.99],[0.271253,-0.225947,-0.523205,-0.775646],[0,1,-1,0],[9E+09,9E+09,9E+09,9E+09,9E+09,9E+09]],s100,z5,a1\WObj:=grinder6;
    MoveL [[-93.65,110.96,-277.99],[0.582497,-0.431583,-0.372192,-0.579574],[0,1,0,0],[9E+09,9E+09,9E+09,9E+09,9E+09,9E+09]],s50,z5,a1\WObj:=grinder6;
    MoveL [[-96.49,104.60,-277.90],[0.495905,-0.539702,-0.494579,-0.46711],[0,0,0,0],[9E+09,9E+09,9E+09,9E+09,9E+09,9E+09]],s50,z5,a1\WObj:=grinder6;
    MoveL [[-92.78,104.61,-277.97],[0.599892,-0.649356,-0.338073,-0.322759],[0,0,0,0],[9E+09,9E+09,9E+09,9E+09,9E+09,9E+09]],s50,z5,a1\WObj:=grinder6;
    MoveL [[-89.97,86.38,-278.00],[0.559521,-0.606973,-0.409387,-0.388486],[0,0,0,0],[9E+09,9E+09,9E+09,9E+09,9E+09,9E+09]],s50,z5,a1\WObj:=grinder6;
    MoveL [[-91.53,120.74,-277.93],[0.56962,-0.617576,-0.393126,-0.37361],[0,0,0,0],[9E+09,9E+09,9E+09,9E+09,9E+09,9E+09]],s50,z5,a1\WObj:=grinder6;
    !
    MoveJ [[-214.39,117.58,-277.90],[0.569607,-0.617542,-0.393141,-0.373671],[0,0,0,0],[9E+09,9E+09,9E+09,9E+09,9E+09,9E+09]],s300,z50,a1\WObj:=grinder6;
    MoveJ [[-273.96,162.51,-278.06],[0.26948,-0.6327,0.664108,0.293312],[1,0,-2,0],[9E+09,9E+09,9E+09,9E+09,9E+09,9E+09]],s500,z50,a1\WObj:=grinder6;
    !
    MoveL [[-114.36,100.45,-278.20],[0.408895,-0.812803,0.393109,0.132747],[1,0,-2,0],[9E+09,9E+09,9E+09,9E+09,9E+09,9E+09]],s300,z50,a1\WObj:=grinder6;
    MoveL [[-88.01,80.15,-278.19],[0.408904,-0.81277,0.393155,0.132782],[1,0,-2,0],[9E+09,9E+09,9E+09,9E+09,9E+09,9E+09]],s100,z5,a1\WObj:=grinder6;
    MoveL [[-84.16,119.19,-278.18],[0.423589,-0.902224,-0.0329732,-0.074003],[1,0,-3,0],[9E+09,9E+09,9E+09,9E+09,9E+09,9E+09]],s50,z5,a1\WObj:=grinder6;
    MoveL [[-93.46,103.17,-295.34],[0.334883,-0.706861,0.561048,0.270973],[1,0,-2,0],[9E+09,9E+09,9E+09,9E+09,9E+09,9E+09]],s50,z5,a1\WObj:=grinder6;
    MoveL [[-96.73,104.62,-295.40],[0.150055,-0.337438,0.828873,0.420225],[1,0,-1,0],[9E+09,9E+09,9E+09,9E+09,9E+09,9E+09]],s50,z5,a1\WObj:=grinder6;
    MoveL [[-98.82,102.54,-295.47],[0.0566992,-0.137037,0.881384,0.448518],[1,0,-1,0],[9E+09,9E+09,9E+09,9E+09,9E+09,9E+09]],s50,z5,a1\WObj:=grinder6;
    MoveL [[-96.88,96.39,-295.45],[0.186243,-0.319028,0.850852,0.373613],[1,0,-1,0],[9E+09,9E+09,9E+09,9E+09,9E+09,9E+09]],s50,z5,a1\WObj:=grinder6;
    MoveL [[-88.66,97.16,-295.38],[0.363861,-0.691295,0.580672,0.229209],[1,0,-2,0],[9E+09,9E+09,9E+09,9E+09,9E+09,9E+09]],s100,z5,a1\WObj:=grinder6;
    MoveL [[-86.96,85.93,-295.37],[0.450252,-0.638401,0.605447,0.152156],[1,0,-2,0],[9E+09,9E+09,9E+09,9E+09,9E+09,9E+09]],s50,z5,a1\WObj:=grinder6;
    MoveL [[-86.97,85.93,-295.38],[0.560112,-0.544532,0.623564,0.030451],[1,1,-2,0],[9E+09,9E+09,9E+09,9E+09,9E+09,9E+09]],s50,z5,a1\WObj:=grinder6;
    MoveL [[-84.99,88.10,-295.48],[0.462646,-0.81178,0.162708,-0.317015],[1,1,-3,0],[9E+09,9E+09,9E+09,9E+09,9E+09,9E+09]],s100,z5,a1\WObj:=grinder6;
    MoveL [[-87.99,92.22,-295.57],[0.495976,-0.862817,0.0333931,-0.0918678],[1,0,-3,0],[9E+09,9E+09,9E+09,9E+09,9E+09,9E+09]],s50,z5,a1\WObj:=grinder6;
    MoveL [[-86.30,76.32,-295.45],[0.543884,-0.711689,0.154539,-0.416901],[1,1,-3,0],[9E+09,9E+09,9E+09,9E+09,9E+09,9E+09]],s50,z5,a1\WObj:=grinder6;
    !
    MoveL [[-158.53,85.50,-319.94],[0.305913,-0.722716,-0.541105,-0.302167],[1,0,-4,0],[9E+09,9E+09,9E+09,9E+09,9E+09,9E+09]],s500,z50,a1\WObj:=grinder6;
    !
    MoveL [[-94.73,99.83,-319.87],[0.350337,-0.799791,-0.41871,-0.249558],[1,0,-3,0],[9E+09,9E+09,9E+09,9E+09,9E+09,9E+09]],s300,z50,a1\WObj:=grinder6;
    MoveL [[-92.52,95.39,-286.22],[0.441241,-0.71825,-0.325093,-0.428647],[0,1,-4,0],[9E+09,9E+09,9E+09,9E+09,9E+09,9E+09]],s100,z50,a1\WObj:=grinder6;
    MoveL [[-91.36,95.39,-260.92],[0.473498,-0.625759,-0.442453,-0.43412],[0,0,-4,0],[9E+09,9E+09,9E+09,9E+09,9E+09,9E+09]],s100,z50,a1\WObj:=grinder6;
    MoveL [[-91.39,95.39,-218.53],[0.447963,-0.599524,-0.477448,-0.460373],[0,0,-4,0],[9E+09,9E+09,9E+09,9E+09,9E+09,9E+09]],s100,z50,a1\WObj:=grinder6;
    MoveL [[-101.66,85.99,-173.13],[0.443221,-0.505863,-0.491577,-0.553181],[0,1,-4,0],[9E+09,9E+09,9E+09,9E+09,9E+09,9E+09]],s100,z50,a1\WObj:=grinder6;
    MoveL [[-112.97,85.99,-157.15],[0.405119,-0.471744,-0.524446,-0.581629],[0,1,-4,0],[9E+09,9E+09,9E+09,9E+09,9E+09,9E+09]],s100,z50,a1\WObj:=grinder6;
    !
    MoveL [[-292.60,34.68,-69.72],[0.345815,-0.455467,-0.64453,-0.507487],[0,0,-4,0],[9E+09,9E+09,9E+09,9E+09,9E+09,9E+09]],s500,z50,a1\WObj:=grinder6;
    MoveL [[-332.45,-137.87,-85.15],[0.52183,-0.843247,0.128273,0.0131596],[0,0,-3,0],[9E+09,9E+09,9E+09,9E+09,9E+09,9E+09]],s500,z50,a1\WObj:=grinder6;
    !!
    S_Grinder6 "Stop";
ENDPROC

ENDMODULE
